///////////////////////////////////////////////////////////////////////////////////////
// ---   Formateo del Evento de Estado del Dispositivo
// ---   * Mirar si hay sitio para generar el nuevo evento
// ---       * Inicializo NumBytes y Puntero al DB de Eventos Generados
// ---       * Calcula el tamaño de bytes que hay en el DB de Eventos Generados
// ---       * Comprobar si hay sitio para un evento más
// ---   *  Formatear el evento de Estado de Inicio de Bucle  INI!
///////////////////////////////////////////////////////////////////////////////////////


///////////////////////////////////////////////////////////////////////////////////////
// --- Mirar si hay sitio para generar un evento más
      L     0;
      T     #NumBytes;  // Inicializo el numero de Bytes
      T     #P_Eventos;  // Inicializo el puntero de Eventos Generados

Inicio_BusquedaFinalEventos_MckeysEnMesa:NOP   0;
      OPN   DB [#DBEventos];  // Calcula el tamaño de bytes que hay en el DB
      L     DBB [#P_Eventos];
      L     0;
      ==I;
      JC    Fin_BusquedaFinalEventos_MckeysEnMesa;  // Buscamos el final del DB = 0

      OPN   DB [#DBEventos];
      L     DBB [#P_Eventos];
      L     ' ';
      ==I;
      JC    Fin_BusquedaFinalEventos_MckeysEnMesa;  // Buscamos el final del DB = ' '

      L     #P_Eventos;  // Incremento de P#1.0
      L     P#1.0;
      +D;
      T     #P_Eventos;

      JU    Inicio_BusquedaFinalEventos_MckeysEnMesa;  // Continuar con el siguiente posicion

Fin_BusquedaFinalEventos_MckeysEnMesa:NOP   0;
      L     #P_Eventos;  // Sacamos el NumBytes Escritos
      SRD   3;
      T     #NumBytes;

      L     #NumBytes;  // Miramos si hay sitio
      L     #MaxBytes;  // Max. que se pueden emitir, parametro
      >I;
      JC    FinalFuncion;  // No se pueden generar más eventos



///////////////////////////////////////////////////////////////////////////////////////
// --- Formatear el evento
      L     #P_Eventos;
      LAR2;  // Puntero al DB de Eventos Generados

      TAR2;  // Mirar si es el primer evento de la lista
      L     0;
      ==I;
      JC    NoEsInicio_ListaDeEventos_MckeysEnMesa;  // Es el primero

      OPN   DB [#DBEventos];
      L     ',';  // Separador entre eventos ','
      T     DBB [AR2, P#0.0];
      +AR2  P#1.0;

NoEsInicio_ListaDeEventos_MckeysEnMesa:NOP   0;

///////////////////////////////////////////////////////////////////////////////
// --- Cuerpo del Evento
      OPN   DB [#DBEventos];  // DB de Eventos Generados (A Emitir)
      L     '{';  // Inicio de Evento '{'
      T     DBB [AR2, P#0.0];
      +AR2  P#1.0;

      L     'CHE!';  // Evento - CHE!
      T     DBD [AR2, P#0.0];
      +AR2  P#4.0;


///////////////////////////////////////////////////////////////////////////////
      L     '[';
      T     DBB [AR2, P#0.0];
      L     'TIPO';
      T     DBD [AR2, P#1.0];
      L     ']';  // Evento - Atributo Mckey '[TIPO]'
      T     DBB [AR2, P#5.0];
      +AR2  P#6.0;

      L     'MESA';
      T     DBD [AR2, P#0.0];
      +AR2  P#4.0;


///////////////////////////////////////////////////////////////////////////////
      OPN   DB [#DBEventos];
      L     '[';  // Evento - Atributo Mesa  '[NUME]'
      T     DBB [AR2, P#0.0];
      L     'NUME';
      T     DBD [AR2, P#1.0];
      L     ']';
      T     DBB [AR2, P#5.0];
      +AR2  P#6.0;

      L     #NumMesa;
      L     "CTE_OffsetMesa";
      +I;
      T     #Valor;

// --- Convertir Valor a ASCII -  Mesa Actual
      TAR2;
      SRD   3;
      T     #NumBytes;  // Miro que offset tiene la String

      CALL  "FC893_Obtener_StringDelAtributo"
      ( DB_String := #NumDBEventos,
        OffsetIni := #NumBytes,
        Valor     := #Valor,
        OffsetFin := #Offset
      );  // Llamo a ObtenerStrinAtributo

      L     #Offset;
      SLD   3;
      LAR2;  // Recupero que offset tiene la String
// --- Ya esta convertido el Valor a ASCI - Fin Mesa Actual



///////////////////////////////////////////////////////////////////////////////
      L     '[';
      T     DBB [AR2, P#0.0];
      L     'OPER';
      T     DBD [AR2, P#1.0];
      L     ']';  // Evento - Atributo Mckey '[TIPO]'
      T     DBB [AR2, P#5.0];
      +AR2  P#6.0;

      L     'MCKY';
      T     DBD [AR2, P#0.0];
      +AR2  P#4.0;


///////////////////////////////////////////////////////////////////////////////
      OPN   DB [#DBEventos];
      L     '[';  // Evento - Atributo Mckeys '[MCKY]'
      T     DBB [AR2, P#0.0];
      L     'MCKY';
      T     DBD [AR2, P#1.0];
      L     ']';
      T     DBB [AR2, P#5.0];
      +AR2  P#6.0;

// ---- Inicio de Mckeys
      OPN   DB [#DBEventos];
      L     '(';
      T     DBB [AR2, P#0.0];
      +AR2  P#1.0;

// --- Bucle de Mckeys >>> Hay Una UT
      L     "DB810_ColasMesas".Colas[#NumMesa].UT_PrimeraMesa;
      T     #NumeroUT;

      SET;  // Hay UT ?
      L     #NumeroUT;
      L     0;
      ==I;
      JC    FinalBucleUTs_MckeysEnMesa;

      L     "DB812_UTs_Control".UT[#NumeroUT].Mckey;
      T     #Valor;

// --- Convertir Valor a ASCII -  Mesa Actual
      TAR2;
      SRD   3;
      T     #NumBytes;  // Miro que offset tiene la String

      CALL  "FC893_Obtener_StringDelAtributo"
      ( DB_String := #NumDBEventos,
        OffsetIni := #NumBytes,
        Valor     := #Valor,
        OffsetFin := #Offset
      );  // Llamo a ObtenerStrinAtributo

      L     #Offset;
      SLD   3;
      LAR2;  // Recupero que offset tiene la String
// --- Ya esta convertido el Valor a ASCI - Fin Mesa Actual

      L     "DB812_UTs_Control".UT[#NumeroUT].UT_SiguienteMesa;
      T     #NumeroUT;

// --- Bucle de Mckeys >>> Hay Mas UTs
IncioBucleUTs_MckeysEnMesa:NOP   0;
      SET;  // Hay UT ?
      L     #NumeroUT;
      L     0;
      ==I;
      JC    FinalBucleUTs_MckeysEnMesa;

      OPN   DB [#DBEventos];
      L     ',';  // Separador de Mckeys
      T     DBB [AR2, P#0.0];
      +AR2  P#1.0;

      L     "DB812_UTs_Control".UT[#NumeroUT].Mckey;
      T     #Valor;

// --- Convertir Valor a ASCII -  Mesa Actual
      TAR2;
      SRD   3;
      T     #NumBytes;  // Miro que offset tiene la String

      CALL  "FC893_Obtener_StringDelAtributo"
      ( DB_String := #NumDBEventos,
        OffsetIni := #NumBytes,
        Valor     := #Valor,
        OffsetFin := #Offset
      );  // Llamo a ObtenerStrinAtributo

      L     #Offset;
      SLD   3;
      LAR2;  // Recupero que offset tiene la String
// --- Ya esta convertido el Valor a ASCI - Fin Mesa Actual


      L     "DB812_UTs_Control".UT[#NumeroUT].UT_SiguienteMesa;
      T     #NumeroUT;
      JU    IncioBucleUTs_MckeysEnMesa;

FinalBucleUTs_MckeysEnMesa:NOP   0;

// --- Final de Mckeys
      OPN   DB [#DBEventos];
      L     ')';
      T     DBB [AR2, P#0.0];
      +AR2  P#1.0;


///////////////////////////////////////////////////////////////////////////////
      OPN   DB [#DBEventos];
      L     '[';  // Evento - Atributo Resultado'[RESU]'
      T     DBB [AR2, P#0.0];
      L     'RESU';
      T     DBD [AR2, P#1.0];
      L     ']';
      T     DBB [AR2, P#5.0];
      +AR2  P#6.0;

      L     'OK';
      T     DBW [AR2, P#0.0];
      +AR2  P#2.0;


///////////////////////////////////////////////////////////////////////////////
// --- Final del Evento

      OPN   DB [#DBEventos];  // DB de Eventos Generados (A Emitir)
      L     '}';  // --- Fin de Evento '}'
      T     DBB [AR2, P#0.0];
      +AR2  P#1.0;


///////////////////////////////////////////////////////////////////////////////
/// -- Dar  por enviado el evento

      SET;
      R     "DB831_Mesas".Mesas[#NumMesa].EventosInformarJdT.MckeysEnMesa;

      JU    Siguiente_BucleDeMesas;



NETWORK
TITLE = Evento de Evento de Todo De Mesa >>> Ocupacion, Mckeys
EnviarEvento_TodoDeMesa:NOP   0;

///////////////////////////////////////////////////////////////////////////////////////
// ---   Formateo del Evento de Estado del Dispositivo
// ---   * Mirar si hay sitio para generar el nuevo evento
// ---       * Inicializo NumBytes y Puntero al DB de Eventos Generados
// ---       * Calcula el tamaño de bytes que hay en el DB de Eventos Generados
// ---       * Comprobar si hay sitio para un evento más
// ---   *  Formatear el evento de Estado de Inicio de Bucle  INI!
///////////////////////////////////////////////////////////////////////////////////////


///////////////////////////////////////////////////////////////////////////////////////
// --- Mirar si hay sitio para generar un evento más
      L     0;
      T     #NumBytes;  // Inicializo el numero de Bytes
      T     #P_Eventos;  // Inicializo el puntero de Eventos Generados

Inicio_BusquedaFinalEventos_TodoDeMesa:NOP   0;
      OPN   DB [#DBEventos];  // Calcula el tamaño de bytes que hay en el DB
      L     DBB [#P_Eventos];
      L     0;
      ==I;
      JC    Fin_BusquedaFinalEventos_TodoDeMesa;  // Buscamos el final del DB = 0

      OPN   DB [#DBEventos];
      L     DBB [#P_Eventos];
      L     ' ';
      ==I;
      JC    Fin_BusquedaFinalEventos_TodoDeMesa;  // Buscamos el final del DB = ' '

      L     #P_Eventos;  // Incremento de P#1.0
      L     P#1.0;
      +D;
      T     #P_Eventos;

      JU    Inicio_BusquedaFinalEventos_TodoDeMesa;  // Continuar con el siguiente posicion

Fin_BusquedaFinalEventos_TodoDeMesa:NOP   0;
      L     #P_Eventos;  // Sacamos el NumBytes Escritos
      SRD   3;
      T     #NumBytes;

      L     #NumBytes;  // Miramos si hay sitio
      L     #MaxBytes;  // Max. que se pueden emitir, parametro
      >I;
      JC    FinalFuncion;  // No se pueden generar más eventos



///////////////////////////////////////////////////////////////////////////////////////
// --- Formatear el evento
      L     #P_Eventos;
      LAR2;  // Puntero al DB de Eventos Generados

      TAR2;  // Mirar si es el primer evento de la lista
      L     0;
      ==I;
      JC    NoEsInicio_ListaDeEventos_TodoDeMesa;  // Es el primero

      OPN   DB [#DBEventos];
      L     ',';  // Separador entre eventos ','
      T     DBB [AR2, P#0.0];
      +AR2  P#1.0;

NoEsInicio_ListaDeEventos_TodoDeMesa:NOP   0;

///////////////////////////////////////////////////////////////////////////////
// --- Cuerpo del Evento
      OPN   DB [#DBEventos];  // DB de Eventos Generados (A Emitir)
      L     '{';  // Inicio de Evento '{'
      T     DBB [AR2, P#0.0];
      +AR2  P#1.0;

      L     'CHE!';  // Evento - CHE!
      T     DBD [AR2, P#0.0];
      +AR2  P#4.0;


///////////////////////////////////////////////////////////////////////////////
      L     '[';
      T     DBB [AR2, P#0.0];
      L     'TIPO';
      T     DBD [AR2, P#1.0];
      L     ']';  // Evento - Atributo Mckey '[TIPO]'
      T     DBB [AR2, P#5.0];
      +AR2  P#6.0;

      L     'MESA';
      T     DBD [AR2, P#0.0];
      +AR2  P#4.0;


///////////////////////////////////////////////////////////////////////////////
      OPN   DB [#DBEventos];
      L     '[';  // Evento - Atributo Mesa  '[NUME]'
      T     DBB [AR2, P#0.0];
      L     'NUME';
      T     DBD [AR2, P#1.0];
      L     ']';
      T     DBB [AR2, P#5.0];
      +AR2  P#6.0;

      L     #NumMesa;
      L     "CTE_OffsetMesa";
      +I;
      T     #Valor;

// --- Convertir Valor a ASCII -  Mesa Actual
      TAR2;
      SRD   3;
      T     #NumBytes;  // Miro que offset tiene la String

      CALL  "FC893_Obtener_StringDelAtributo"
      ( DB_String := #NumDBEventos,
        OffsetIni := #NumBytes,
        Valor     := #Valor,
        OffsetFin := #Offset
      );  // Llamo a ObtenerStrinAtributo

      L     #Offset;
      SLD   3;
      LAR2;  // Recupero que offset tiene la String
// --- Ya esta convertido el Valor a ASCI - Fin Mesa Actual



///////////////////////////////////////////////////////////////////////////////
      L     '[';
      T     DBB [AR2, P#0.0];
      L     'OPER';
      T     DBD [AR2, P#1.0];
      L     ']';  // Evento - Atributo Mckey '[TIPO]'
      T     DBB [AR2, P#5.0];
      +AR2  P#6.0;

      L     'TODO';
      T     DBD [AR2, P#0.0];
      +AR2  P#4.0;


///////////////////////////////////////////////////////////////////////////////
      OPN   DB [#DBEventos];
      L     '[';  // Evento - Atributo Mckeys '[MCKY]'
      T     DBB [AR2, P#0.0];
      L     'MCKY';
      T     DBD [AR2, P#1.0];
      L     ']';
      T     DBB [AR2, P#5.0];
      +AR2  P#6.0;

// ---- Inicio de Mckeys
      OPN   DB [#DBEventos];
      L     '(';
      T     DBB [AR2, P#0.0];
      +AR2  P#1.0;

// --- Bucle de Mckeys >>> Hay Una UT
      L     "DB810_ColasMesas".Colas[#NumMesa].UT_PrimeraMesa;
      T     #NumeroUT;

      SET;  // Hay UT ?
      L     #NumeroUT;
      L     0;
      ==I;
      JC    FinalBucleUTs_TodoDeMesa;

      L     "DB812_UTs_Control".UT[#NumeroUT].Mckey;
      T     #Valor;

// --- Convertir Valor a ASCII -  Mesa Actual
      TAR2;
      SRD   3;
      T     #NumBytes;  // Miro que offset tiene la String

      CALL  "FC893_Obtener_StringDelAtributo"
      ( DB_String := #NumDBEventos,
        OffsetIni := #NumBytes,
        Valor     := #Valor,
        OffsetFin := #Offset
      );  // Llamo a ObtenerStrinAtributo

      L     #Offset;
      SLD   3;
      LAR2;  // Recupero que offset tiene la String
// --- Ya esta convertido el Valor a ASCI - Fin Mesa Actual

      L     "DB812_UTs_Control".UT[#NumeroUT].UT_SiguienteMesa;
      T     #NumeroUT;

// --- Bucle de Mckeys >>> Hay Mas UTs
IncioBucleUTs_TodoDeMesa:NOP   0;
      SET;  // Hay UT ?
      L     #NumeroUT;
      L     0;
      ==I;
      JC    FinalBucleUTs_TodoDeMesa;

      OPN   DB [#DBEventos];
      L     ',';  // Separador de Mckeys
      T     DBB [AR2, P#0.0];
      +AR2  P#1.0;

      L     "DB812_UTs_Control".UT[#NumeroUT].Mckey;
      T     #Valor;

// --- Convertir Valor a ASCII -  Mesa Actual
      TAR2;
      SRD   3;
      T     #NumBytes;  // Miro que offset tiene la String

      CALL  "FC893_Obtener_StringDelAtributo"
      ( DB_String := #NumDBEventos,
        OffsetIni := #NumBytes,
        Valor     := #Valor,
        OffsetFin := #Offset
      );  // Llamo a ObtenerStrinAtributo

      L     #Offset;
      SLD   3;
      LAR2;  // Recupero que offset tiene la String
// --- Ya esta convertido el Valor a ASCI - Fin Mesa Actual


      L     "DB812_UTs_Control".UT[#NumeroUT].UT_SiguienteMesa;
      T     #NumeroUT;
      JU    IncioBucleUTs_TodoDeMesa;

FinalBucleUTs_TodoDeMesa:NOP   0;





// --- Final de Mckeys
      OPN   DB [#DBEventos];
      L     ')';
      T     DBB [AR2, P#0.0];
      +AR2  P#1.0;


///////////////////////////////////////////////////////////////////////////////
      OPN   DB [#DBEventos];
      L     '[';  // Evento - Atributo Ocupacion '[OCUP]'
      T     DBB [AR2, P#0.0];
      L     'OCUP';
      T     DBD [AR2, P#1.0];
      L     ']';
      T     DBB [AR2, P#5.0];
      +AR2  P#6.0;

      L     'NO';  // No Ocupado

      SET;
      AN    "DB900_Estado_Mesas".EstadoVI[#NumMesa].En_PHS_1;
      AN    "DB900_Estado_Mesas".EstadoVI[#NumMesa].En_PHS_2;
      JC    NoOcupado_TodoDeMesa;

      L     'SI';  // Esta Ocupado

NoOcupado_TodoDeMesa:NOP   0;
      OPN   DB [#DBEventos];
      T     DBW [AR2, P#0.0];
      +AR2  P#2.0;


///////////////////////////////////////////////////////////////////////////////
      OPN   DB [#DBEventos];
      L     '[';  // Evento - Atributo Resultado'[RESU]'
      T     DBB [AR2, P#0.0];
      L     'RESU';
      T     DBD [AR2, P#1.0];
      L     ']';
      T     DBB [AR2, P#5.0];
      +AR2  P#6.0;

      L     'OK';
      T     DBW [AR2, P#0.0];
      +AR2  P#2.0;


///////////////////////////////////////////////////////////////////////////////
// --- Final del Evento

      OPN   DB [#DBEventos];  // DB de Eventos Generados (A Emitir)
      L     '}';  // --- Fin de Evento '}'
      T     DBB [AR2, P#0.0];
      +AR2  P#1.0;


///////////////////////////////////////////////////////////////////////////////
/// -- Dar  por enviado el evento

      SET;
      R     "DB831_Mesas".Mesas[#NumMesa].EventosInformarJdT.TodoDeMesa;

      JU    Siguiente_BucleDeMesas;



NETWORK
TITLE = Emision de Evento Rearme
EnviarEvento_rearme:NOP   0;

///////////////////////////////////////////////////////////////////////////////////////
// ---   Formateo del Evento de Estado del Dispositivo
// ---   * Mirar si hay sitio para generar el nuevo evento
// ---       * Inicializo NumBytes y Puntero al DB de Eventos Generados
// ---       * Calcula el tamaño de bytes que hay en el DB de Eventos Generados
// ---       * Comprobar si hay sitio para un evento más
// ---   *  Formatear el evento de Estado de Inicio de Bucle
///////////////////////////////////////////////////////////////////////////////////////

// --- Primero miramos si tenemos configurado emitir el evento o no
      SET;
      A     "DB831_Mesas".Mesas[#NumMesa].EventosInformarJdT.Evento_Rearme;
      JC    emite_evento_rearme;

      SET;
      R     "DB831_Mesas".Mesas[#NumMesa].Memorias.Evento_rearme;
      JC    Siguiente_BucleDeMesas;

///////////////////////////////////////////////////////////////////////////////////////
// --- Mirar si hay sitio para generar un evento más
emite_evento_rearme:NOP   0;
      L     0;
      T     #NumBytes;  // Inicializo el numero de Bytes
      T     #P_Eventos;  // Inicializo el puntero de Eventos Generados

Inicio_BusquedaFinalEventos_rearme:NOP   0;
      OPN   DB [#DBEventos];  // Calcula el tamaño de bytes que hay en el DB
      L     DBB [#P_Eventos];
      L     0;
      ==I;
      JC    Fin_BusquedaFinalEventos_rearme;  // Buscamos el final del DB = 0

      OPN   DB [#DBEventos];
      L     DBB [#P_Eventos];
      L     ' ';
      ==I;
      JC    Fin_BusquedaFinalEventos_rearme;  // Buscamos el final del DB = ' '

      L     #P_Eventos;  // Incremento de P#1.0
      L     P#1.0;
      +D;
      T     #P_Eventos;

      JU    Inicio_BusquedaFinalEventos_rearme;  //Continuar con el siguiente posicion

Fin_BusquedaFinalEventos_rearme:NOP   0;
      L     #P_Eventos;  // Sacamos el NumBytes Escritos
      SRD   3;
      T     #NumBytes;

      L     #NumBytes;  // Miramos si hay sitio
      L     #MaxBytes;  // Max. que se pueden emitir, parametro
      >I;
      JC    FinalFuncion;  // No se pueden generar más eventos



///////////////////////////////////////////////////////////////////////////////////////
// --- Formatear el evento
      L     #P_Eventos;
      LAR2;  // Puntero al DB de Eventos Generados

      TAR2;  // Mirar si es el primer evento de la lista
      L     0;
      ==I;
      JC    NoEsInicio_ListaDeEventos_rearme;  // Es el primero

      OPN   DB [#DBEventos];
      L     ',';  // Separador entre eventos ','
      T     DBB [AR2, P#0.0];
      +AR2  P#1.0;

NoEsInicio_ListaDeEventos_rearme:NOP   0;

///////////////////////////////////////////////////////////////////////////////
// --- Cuerpo del Evento
      OPN   DB [#DBEventos];  // DB de Eventos Generados (A Emitir)
      L     '{';  // Inicio de Evento '{'
      T     DBB [AR2, P#0.0];
      +AR2  P#1.0;

      L     'EVEN';  // Evento - EVEN
      T     DBD [AR2, P#0.0];
      +AR2  P#4.0;


///////////////////////////////////////////////////////////////////////////////
      L     '[';
      T     DBB [AR2, P#0.0];
      L     'TIPO';
      T     DBD [AR2, P#1.0];
      L     ']';  // Evento - Atributo Mckey '[TIPO]'
      T     DBB [AR2, P#5.0];
      +AR2  P#6.0;

      L     'MESA';
      T     DBD [AR2, P#0.0];
      +AR2  P#4.0;


///////////////////////////////////////////////////////////////////////////////
      OPN   DB [#DBEventos];
      L     '[';  // Evento - Atributo Mesa  '[NUME]'
      T     DBB [AR2, P#0.0];
      L     'NUME';
      T     DBD [AR2, P#1.0];
      L     ']';
      T     DBB [AR2, P#5.0];
      +AR2  P#6.0;

      L     #NumMesa;
      L     "CTE_OffsetMesa";
      +I;
      T     #Valor;

// --- Convertir Valor a ASCII -  Mesa Actual
      TAR2;
      SRD   3;
      T     #NumBytes;  // Miro que offset tiene la String

      CALL  "FC893_Obtener_StringDelAtributo"
      ( DB_String := #NumDBEventos,
        OffsetIni := #NumBytes,
        Valor     := #Valor,
        OffsetFin := #Offset
      );  // Llamo a ObtenerStrinAtributo

      L     #Offset;
      SLD   3;
      LAR2;  // Recupero que offset tiene la String
// --- Ya esta convertido el Valor a ASCI - Fin Mesa Actual



///////////////////////////////////////////////////////////////////////////////
      L     '[';
      T     DBB [AR2, P#0.0];
      L     'OPER';
      T     DBD [AR2, P#1.0];
      L     ']';  // Evento - Atributo Mckey '[TIPO]'
      T     DBB [AR2, P#5.0];
      +AR2  P#6.0;

      L     'REAR';
      T     DBD [AR2, P#0.0];
      +AR2  P#4.0;


///////////////////////////////////////////////////////////////////////////////
// --- Final del Evento

      OPN   DB [#DBEventos];  // DB de Eventos Generados (A Emitir)
      L     '}';  // --- Fin de Evento '}'
      T     DBB [AR2, P#0.0];
      +AR2  P#1.0;


///////////////////////////////////////////////////////////////////////////////
/// -- Dar  por enviado el evento

      SET;
      R     "DB831_Mesas".Mesas[#NumMesa].Memorias.Evento_rearme;

      JU    Siguiente_BucleDeMesas;



NETWORK
TITLE = Final de la Función
/////////////////////////////////////////////////////////////////////////////////////
FinalFuncion:NOP   0;


END_FUNCTION

FUNCTION "FC700_JDT02ControlTracking" : Void   // FC700, LAD
{ S7_Optimized_Access := 'FALSE' }
AUTHOR : TRACKING
NAME : 20141014
VERSION : 4.0
// stored: AutoNumber false, SetENOAutomatically false
BEGIN

NETWORK
TITLE = Previo
// -----------------------------------------------------------------------
// --- Inicialializacion
// --- Borrado de la Base de Datosç

      CALL  "FC701_JDT02ControlCOM";  // Control del Puerto
      CALL  "FC706_JDT02Borrado";



NETWORK
TITLE = Control del Sistema
// ---------------------------------------------------------------------
// --- Control de Recepcion de Eventos

      CALL  "FC702_JDT02RecJdTMensaje";
      CALL  "FC704_JDT02AnalisisRecibidos";
      CALL  "FC810_EventosRecibidos"
      ( NumJDT := 2
      );


// ---------------------------------------------------------------------
// --- Control de EmisionEventos de Eventos

      CALL  "FC811_EventosGenerados"
      ( NumJdT := 2
      );
      CALL  "FC705_JDT02AnalisisEnviados";
      CALL  "FC703_JDT02EmiJdTMensaje";


// ---------------------------------------------------------------------
// --- Control de EmisionEventos de Router
//     *  Proceso Inicialización bucle
//     *  Eventos de la Pantalla (Movimientos)
//     *  Eventos de Reset V2.0   >>> 2023 01 05

//      CALL  "FC816_EventosEnv_Router"
//         NumJDT :=2

// NIEVES 10/04/25
      CALL  "FC717_Emision_Routing"
      ( NumJDT := 2
      );


      CALL  "FC815_EventosEnv_Control"
      ( NumJDT := 2
      );
      CALL  "FC817_EventosEnv_Reset"
      ( NumJDT := 2
      );


Fin:  NOP   0;


END_FUNCTION

FUNCTION "FC701_JDT02ControlCOM" : Void   // FC701, LAD
TITLE = "ControlCOM" - Control de Comunicaciones
{ S7_Optimized_Access := 'FALSE' }
AUTHOR : TRACKING
NAME : 20150129
VERSION : 3.1
// - Contorol y valida el Enlace entre el PLC y el PC
// - Varible: EnlaceCP_OK
// stored: AutoNumber false, SetENOAutomatically false
   VAR_TEMP
      Temporal : Struct   // Temporal para el tratamiento de Result 01
         "0.0" : Bool;
         "0.1" : Bool;
         "0.2" : Bool;
         "0.3" : Bool;
         "0.4" : Bool;
         "0.5" : Bool;
         "0.6" : Bool;
         "0.7" : Bool;
         "1.0" : Bool;
         "1.1" : Bool;
         "1.2" : Bool;
         "1.3" : Bool;
         "1.4" : Bool;
         "1.5" : Bool;
         "1.6" : Bool;
         "1.7" : Bool;
         "2.0" : Bool;
         "2.1" : Bool;
         "2.2" : Bool;
         "2.3" : Bool;
         "2.4" : Bool;
         "2.5" : Bool;
         "2.6" : Bool;
         "2.7" : Bool;
         "3.0" : Bool;
         "3.1" : Bool;
         "3.2" : Bool;
         "3.4" : Bool;
         "3.5" : Bool;
         "3.6" : Bool;
         "3.7" : Bool;
      END_STRUCT;
      P_Temporal : DWord;
      TMPEnlace_OK : Bool;
   END_VAR
BEGIN

NETWORK
TITLE = Control del Enlace - Puerto 2001
// - Distribución  - Conexion  - Desconesion  - Final    ------------------------------------------------------------------------------------------------------   Control del Enlace - Distribución   --- Si hay que desconetar   --- Si esta conectado
      A     "DB701_JDT02StatusCOM".CNTRL_Reset;  // Si hay que desconectar
      O     "DB701_JDT02StatusCOM".RecJdT_Reset;
      O     "DB701_JDT02StatusCOM".EmiJdT_Reset;
      JC    DesConectar;

      A     "DB701_JDT02StatusCOM".EnlaceCP_OK;  // Si está conectado
      JC    Final;

      JU    Conectar;  // Hay que conectar

// ------------------------------------------------------------------------------------------------------
// Control del Enlace - Conexion
// --- Mirar si hay que activar Flanco
// --- Mirar si hay petición de conexion activa
// --- Llamada de Conexion
// --- Comprobación de la Conexion

Conectar:NOP   0;
      AN    "DB891_VariablesTCP".TCON_JdT_PLC_Busy_JDT02;
      AN    "DB891_VariablesTCP".TCON_JdT_PLC_Req_JDT02;
      AN    "DB891_VariablesTCP".TCON_JdT_PLC_Flanco_JDT02;
      =     "DB891_VariablesTCP".TCON_JdT_PLC_Flanco_JDT02;  // -- Activar flanco

      A     "DB891_VariablesTCP".TCON_JdT_PLC_Flanco_JDT02;
      AN    "DB891_VariablesTCP".TCON_JdT_PLC_Req_JDT02;
      S     "DB891_VariablesTCP".TCON_JdT_PLC_Req_JDT02;
      R     "DB891_VariablesTCP".TDISCON_JdT_PLC_Req_JDT02;  // -- Petición de Conexion Activa

      CALL  TCON, "DB896_TCON_JdT_PLC_JDT02"
      ( REQ     := "DB891_VariablesTCP".TCON_JdT_PLC_Flanco_JDT02,
        ID      := W#16#3,
        DONE    := "DB891_VariablesTCP".TCON_JdT_PLC_Done_JDT02,
        BUSY    := "DB891_VariablesTCP".TCON_JdT_PLC_Busy_JDT02,
        ERROR   := "DB891_VariablesTCP".TCON_JdT_PLC_Error_JDT02,
        STATUS  := "DB891_VariablesTCP".TCON_JdT_PLC_Status_JDT02,
        CONNECT := "DB700_JDTD02ConfigEnlace"
      );


      A     "DB891_VariablesTCP".TCON_JdT_PLC_Done_JDT02;  // -- Comprobacion de la Conexion
      R     "DB891_VariablesTCP".TCON_JdT_PLC_Req_JDT02;
      S     "DB701_JDT02StatusCOM".EnlaceCP_OK;

      A     "DB891_VariablesTCP".TCON_JdT_PLC_Error_JDT02;  // -- Error en conexion
      R     "DB891_VariablesTCP".TCON_JdT_PLC_Req_JDT02;

      A     "DB891_VariablesTCP".TCON_JdT_PLC_Req_JDT02;  // --- Control de Bloqueo
      AN    "DB891_VariablesTCP".TCON_JdT_PLC_Busy_JDT02;
      R     "DB891_VariablesTCP".TCON_JdT_PLC_Req_JDT02;

      JU    Final;  // Fin de la Conexión

// ------------------------------------------------------------------------------------------------------
// Control del Enlace - Desconexion
// --- Mirar si hay que activar Flanco
// --- Mirar si hay petición de desconexion activa
// --- Llamada de DesConexion
// --- Comprobación de la DesConexion

DesConectar:SET;
      R     "DB701_JDT02StatusCOM".EnlaceCP_OK;

      AN    "DB891_VariablesTCP".TDISCON_JdT_PLC_Busy_JDT02;
      AN    "DB891_VariablesTCP".TDISCON_JdT_PLC_Req_JDT02;
      AN    "DB891_VariablesTCP".TDISCON_JdT_PLC_Flanco_JDT02;
      =     "DB891_VariablesTCP".TDISCON_JdT_PLC_Flanco_JDT02;  // -- Activar Flanco


      A     "DB891_VariablesTCP".TDISCON_JdT_PLC_Flanco_JDT02;
      AN    "DB891_VariablesTCP".TDISCON_JdT_PLC_Req_JDT02;
      S     "DB891_VariablesTCP".TDISCON_JdT_PLC_Req_JDT02;
      R     "DB891_VariablesTCP".TCON_JdT_PLC_Req_JDT02;  // -- Petición de DesConexion Activa

      CALL  TDISCON, "DB897_TDISCON_JdT_PLC_JDT02"
      ( REQ    := "DB891_VariablesTCP".TDISCON_JdT_PLC_Flanco_JDT02,
        ID     := W#16#3,
        DONE   := "DB891_VariablesTCP".TDISCON_JdT_PLC_Done_JDT02,
        BUSY   := "DB891_VariablesTCP".TDISCON_JdT_PLC_Busy_JDT02,
        ERROR  := "DB891_VariablesTCP".TDISCON_JdT_PLC_Error_JDT02,
        STATUS := "DB891_VariablesTCP".TDISCON_JdT_PLC_Status_JDT02
      );



      A     "DB891_VariablesTCP".TDISCON_JdT_PLC_Done_JDT02;  // -- Comprobacion de la DesConexión
      R     "DB891_VariablesTCP".TDISCON_JdT_PLC_Req_JDT02;


      R     "DB701_JDT02StatusCOM".CNTRL_Reset;
      R     "DB701_JDT02StatusCOM".RecJdT_Reset;
      R     "DB701_JDT02StatusCOM".EmiJdT_Reset;

      A     "DB891_VariablesTCP".TDISCON_JdT_PLC_Error_JDT02;  // -- Error en la DesConexion
      R     "DB891_VariablesTCP".TDISCON_JdT_PLC_Req_JDT02;

      O(;
      L     "DB891_VariablesTCP".TDISCON_JdT_PLC_Status_JDT02;
      L     W#16#80A3;  //Se está intentando deshacer una conexión no existente
      ==I;
      );
      O(;
      L     "DB891_VariablesTCP".TDISCON_JdT_PLC_Status_JDT02;
      L     W#16#8086;  //El parámetro ID se encuentra en un rango no permitido
      ==I;
      );
      R     "DB891_VariablesTCP".TDISCON_JdT_PLC_Busy_JDT02;
      R     "DB891_VariablesTCP".TDISCON_JdT_PLC_Req_JDT02;
      R     "DB891_VariablesTCP".TDISCON_JdT_PLC_Flanco_JDT02;

      A     "DB891_VariablesTCP".TDISCON_JdT_PLC_Req_JDT02;  // --- Control de Bloqueo
      AN    "DB891_VariablesTCP".TDISCON_JdT_PLC_Busy_JDT02;
      R     "DB891_VariablesTCP".TDISCON_JdT_PLC_Req_JDT02;

      R     "DB701_JDT02StatusCOM".CNTRL_Reset;
      R     "DB701_JDT02StatusCOM".RecJdT_Reset;
      R     "DB701_JDT02StatusCOM".EmiJdT_Reset;

      JU    Final;  // Fin de la DesConexión

// ------------------------------------------------------------------------------------------------------
// Control del Enlace - Final

Final:NOP   0;


END_FUNCTION

FUNCTION "FC706_JDT02Borrado" : Void   // FC706, LAD
TITLE = "BorrodoTracking" - Borrado de toda la Base de Datos
{ S7_Optimized_Access := 'FALSE' }
AUTHOR : TRACKING
NAME : 20130301
VERSION : 3.0
// - Borrado de todos los DB's
// - Inicializadcion del DB de DatosUT
// stored: AutoNumber false, SetENOAutomatically false
   VAR_TEMP
      NumeroUT : Int;
      NumDB : Word;
      UTVacia : Int;
   END_VAR
BEGIN

NETWORK
TITLE = Borrado de todos los DB's de Comunicacion
// -------------------------------------------------------------------------------
// --- Mirar si hay que resetear
      AN    "DB701_JDT02StatusCOM".ResetBD;
      JC    NoResetear;

// -------------------------------------------------------------------------------
// Borrado de los DB de Recepcion de Eventos

      CALL  "FC898_BorrarMensaje"
      ( DB_A_RESET := "DB702_JDT02RecepMensaje"
      );
      CALL  "FC898_BorrarMensaje"
      ( DB_A_RESET := "DB704_JDT02UltimoRecibido"
      );
      CALL  "FC898_BorrarMensaje"
      ( DB_A_RESET := "DB708_JDT02EventosRecibidos"
      );

// -------------------------------------------------------------------------------
// Borrado de los DB de Emision de Eventos

      CALL  "FC898_BorrarMensaje"
      ( DB_A_RESET := "DB703_JDT02EmisionMensaje"
      );
      CALL  "FC898_BorrarMensaje"
      ( DB_A_RESET := "DB705_JDT02UltimoEnviado"
      );
      CALL  "FC898_BorrarMensaje"
      ( DB_A_RESET := "DB706_JDT02EmisionAK"
      );
      CALL  "FC898_BorrarMensaje"
      ( DB_A_RESET := "DB707_JDT02EventosGenerados"
      );

// -------------------------------------------------------------------------------
// Borrado de los DB de la BD de Mesas
// El DB de CrucesMesas no se borra, esto es fijo para cada instalación

      CALL  "FC898_BorrarMensaje"
      ( DB_A_RESET := "DB810_ColasMesas"
      );
      CALL  "FC898_BorrarMensaje"
      ( DB_A_RESET := "DB811_ColasMckeys"
      );

      CALL  "FC898_BorrarMensaje"
      ( DB_A_RESET := "DB812_UTs_Control"
      );
      CALL  "FC898_BorrarMensaje"
      ( DB_A_RESET := "DB813_UTs_Ruta"
      );

      CALL  "FC898_BorrarMensaje"
      ( DB_A_RESET := "DB814_UTs_Etiqueta"
      );
      CALL  "FC898_BorrarMensaje"
      ( DB_A_RESET := "DB815_UTs_Datos"
      );
      CALL  "FC898_BorrarMensaje"
      ( DB_A_RESET := "DB816_UTs_TextoPantalla"
      );
      CALL  "FC898_BorrarMensaje"
      ( DB_A_RESET := "DB820_UTs_DatosQUBIQA"
      );
      CALL  "FC898_BorrarMensaje"
      ( DB_A_RESET := "DB821_UTs_DatosIKPAL"
      );


// -------------------------------------------------------------------------------
// Borrado de los DB de la BD de Dispositivos

      CALL  "FC898_BorrarMensaje"
      ( DB_A_RESET := "DB830_Dispositivos"
      );
      CALL  "FC898_BorrarMensaje"
      ( DB_A_RESET := "DB831_Mesas"
      );
      CALL  "FC898_BorrarMensaje"
      ( DB_A_RESET := "DB832_Maquinas"
      );


// -------------------------------------------------------------------------------
// Borrado de los DB Emision y Recepcion con la instalación

      CALL  "FC898_BorrarMensaje"
      ( DB_A_RESET := "DB840_Emision"
      );
      CALL  "FC898_BorrarMensaje"
      ( DB_A_RESET := "DB841_Recepcion"
      );
      CALL  "FC898_BorrarMensaje"
      ( DB_A_RESET := "DB843_RecepcionPantalla"
      );

      SET;
      R     "DB701_JDT02StatusCOM".ResetBD;

      JU    FinFuncion;  // El siguiente segmento no se realiza


NETWORK
TITLE = ----
// Se acabo la inicializacion
NoResetear:NOP   0;
      L     0;
      LAR1;

// -------------------------------------------------------------------------------
// Borrado de los DB de Recepcion de Eventos, si es necesario

      OPN   "DB702_JDT02RecepMensaje";
      L     DBB [AR1, P#0.0];
      L     ' ';
      <>I;
      JC    S_31;
      CALL  "FC898_BorrarMensaje"
      ( DB_A_RESET := "DB702_JDT02RecepMensaje"
      );

S_31: OPN   "DB704_JDT02UltimoRecibido";
      L     DBB [AR1, P#0.0];
      L     ' ';
      <>I;
      JC    S_32;
      CALL  "FC898_BorrarMensaje"
      ( DB_A_RESET := "DB704_JDT02UltimoRecibido"
      );

S_32: OPN   "DB708_JDT02EventosRecibidos";
      L     DBB [AR1, P#0.0];

      L     ' ';
      <>I;
      JC    S_33;
      CALL  "FC898_BorrarMensaje"
      ( DB_A_RESET := "DB708_JDT02EventosRecibidos"
      );

// -------------------------------------------------------------------------------
// Borrado de los DB de Emision de Eventos, si es necesario

S_33: OPN   "DB703_JDT02EmisionMensaje";
      L     DBB [AR1, P#0.0];
      L     ' ';
      <>I;
      JC    S_34;
      CALL  "FC898_BorrarMensaje"
      ( DB_A_RESET := "DB703_JDT02EmisionMensaje"
      );

S_34: OPN   "DB705_JDT02UltimoEnviado";
      L     DBB [AR1, P#0.0];
      L     ' ';
      <>I;
      JC    S_35;
      CALL  "FC898_BorrarMensaje"
      ( DB_A_RESET := "DB705_JDT02UltimoEnviado"
      );

S_35: OPN   "DB706_JDT02EmisionAK";
      L     DBB [AR1, P#0.0];
      L     ' ';
      <>I;
      JC    S_36;
      CALL  "FC898_BorrarMensaje"
      ( DB_A_RESET := "DB706_JDT02EmisionAK"
      );

S_36: OPN   "DB707_JDT02EventosGenerados";
      L     DBB [AR1, P#0.0];
      L     ' ';
      <>I;
      JC    S_39;
      CALL  "FC898_BorrarMensaje"
      ( DB_A_RESET := "DB707_JDT02EventosGenerados"
      );

S_39: NOP   0;
      JU    FinFuncion;


NETWORK
TITLE = Final de la funcion
FinFuncion:NOP   0;



END_FUNCTION

FUNCTION "FC704_JDT02AnalisisRecibidos" : Void   // FC704, LAD
TITLE = "AnalisisRecibidos" - Analizar los mensajes recibidos por TCP/IP
{ S7_Optimized_Access := 'FALSE' }
AUTHOR : TRACKING
NAME : 20141014
VERSION : 4.0
// - Analizar si el mensaje en si es correcto
// - Distribución
//    - Mensaje ACKN (Validar ID)
//    - Mensaje PING
//    - Resto de mensajes (Validar ID)
// stored: AutoNumber false, SetENOAutomatically false
   VAR_TEMP
      Longitud : UDInt;   // Longitud del Mensaje
      IDMensaje : UDInt;   // ID del Mensaje Recibido
      IniListaEventos : DWord;   // Puntero donde empieza la lista de los eventos
      BytesListaEventos : UDInt;   // Numero de bytes que tiene la lista de los eventos
      DBUltimoRec : Word;   // DB del Ultimo Mensaje Recibido
      DBUltimoEmi : Word;   // DB del Ultimo Mensaje Enviado
      DBEventosRec : Word;   // DB de lista de Eventos Recibidos
      DBEmiAK : Word;   // DB de Emision del Evento AK - Confirmacion
      ReturnValor : Int;   // Temporal
      POrigen : Any;   // Puntero ANY del Origen
      PDestino : Any;   // Puntero ANY del Destino
      IdentEmisor : DWord;
      IdentReceptor : DWord;
      TMPEsperaKA : UDInt;
   END_VAR
BEGIN

NETWORK
TITLE = Inicializamos
// - Inicializaciones de las variables de los DB
// - Coger de la configuracion el Identificador del Emisor (12)
// - Coger de la configuracion el Identificador del Receptor (18)
// -------------------------------------------------------------------------------------------
// Si trabaja sin Agencia  2018 01 24
      SET;
      AN    "Activar_JDT02";  // Mirar si se trabaja con agencia
      JC    Final;

// --------------------------------------------------------------------------------------------
// Inicializaciones de las variables de los DB

      L     "JDT2_NDB_UltimoRec";  // Cogemos el DB de UltimoRecibido
      T     #DBUltimoRec;
      L     "JDT2_NDB_EventosRec";  // Cogemos el DB de EventosRecibidos
      T     #DBEventosRec;

      L     "JDT2_NDB_AKEmi";  // Cogemos el DB de EmisionAK
      T     #DBEmiAK;
      L     "JDT2_NDB_UltimoEmi";  // Cogemos el DB de UltimoEnviado
      T     #DBUltimoEmi;


// --------------------------------------------------------------------------------------------
// Coger de la configuracion el Idendificador del emisor

      L     "JDT2_IdentEmisor";
      T     #IdentEmisor;

// --------------------------------------------------------------------------------------------
// Coger de la configuracion el Idendificador del receptor

      L     "JDT2_IdentReceptor";
      T     #IdentReceptor;


NETWORK
TITLE = Comprobación de la consistencia del mensaje
// Mirar si es correcto
// - Si es Inicio del Mensaje
// - Si es Fin del Mensaje
// - Si es Correcto el Destinario del Mensaje
// - Si es Correcto el Origen del Mensaje
// --------------------------------------------------------------------------------------------
// Mirar si hay mensaje

      L     0;  // Preparar el puntero al Primer byte
      LAR1;
      OPN   DB [#DBUltimoRec];
      L     DBB [AR1, P#0.0];  // Si hay mensaje a tratar <> 0 el primer byte
      L     0;
      ==I;
      JC    Final;  // No hay mensaje

// --------------------------------------------------------------------------------------------
// 1º Paso - Comprobación de que existe Inicio de Mensaje

      OPN   DB [#DBUltimoRec];
      L     DBB [AR1, P#0.0];  // Inicio de Mensaje debe ser 0x02
      L     2;
      ==I;
      JCN   ErrorDeMensajeRecibido;  // Error de Mensaje, Inicio NOK

// --------------------------------------------------------------------------------------------
// 2º Paso - Comprobación de que existe Final del Mensaje

      CALL  "FC890_EtiqChar_EtiqDInt"
      ( DB_String   := "JDT2_NDB_UltimoRec",  // DB del UltimoRecibido
        Long_String := 5,
        Offset_Ini  := 20,
        Valor       := #Longitud
      );  // Calcular la longitud del mensaje

      L     #Longitud;  // Preparar el puntero
      L     1;
      -D;
      SLD   3;
      LAR1;
      OPN   DB [#DBUltimoRec];  // Fin de Mensaje debe ser 0x03
      L     DBB [AR1, P#0.0];
      L     3;
      ==I;
      JCN   ErrorDeMensajeRecibido;  // Error de Mensaje, Fin NOK

// --------------------------------------------------------------------------------------------
// 3º Paso - Comprobación del Emisor del  Mensaje

      L     0;  // Preparar Puntero
      LAR1;
      OPN   DB [#DBUltimoRec];
      L     DBD [AR1, P#6.0];  // Comprobacion del Emisor
      L     #IdentReceptor;
      <>D;
      JC    ErrorDeMensajeRecibido;  // Error de Mensaje, Emisor NOK

// --------------------------------------------------------------------------------------------
// 4º Paso - Comprobación del Receptor del  Mensaje

      OPN   DB [#DBUltimoRec];
      L     DBD [AR1, P#11.0];  // Comprobación del Receptor
      L     #IdentEmisor;
      <>D;
      JC    ErrorDeMensajeRecibido;  // Error de Mensaje, Receptor NOK


NETWORK
TITLE = Distribucion
// - Mirar si es mensaje ACKN - Confirmacion
// - Mirar si es mensaje PING - Keep Alive
// - Es Mensaje de Evento
// --------------------------------------------------------------------------------------------
// 1º Paso - Mirar si es Mensaje AK

      L     0;  // Preparar puntero
      LAR1;
      OPN   DB [#DBUltimoRec];
      L     DBD [AR1, P#24.0];
      L     'ACKN';
      ==I;
      JC    MensajeRecibido_AcuseDeRecibo;  // Recibido Mensaje ACKN - Confirmacion

// --------------------------------------------------------------------------------------------
// 2º Paso - Mirar si es Mensaje KA

      OPN   DB [#DBUltimoRec];
      L     DBD [AR1, P#24.0];
      L     'PING';
      ==I;
      JC    MensajeRecibido_KeepAlive;  // Recibido Mensaje PING - Keep Alive

// --------------------------------------------------------------------------------------------
// 3º Paso - Es Mensaje Evento

      JU    MensajeRecibido_ListaDeEventos;  // Otro tipo de Evento


NETWORK
TITLE = Recibido Mensaje ACKN - Confirmacion del Mensaje Enviado
// - Mirar si esta esperando el Mensaje ACKN - Confirmacion
// - Comprobacion del ID del Mensaje
// - Si es el mismo Numero Secuencial dar por envioado el Mensaje
// - Resetear la variable del Timer Keep Alive y Borrar Mensaje Tratado
// --------------------------------------------------------------------------------------------
// 1º Paso - Comprobamos si esta esperando el Mensaje
MensajeRecibido_AcuseDeRecibo:NOP   0;

      L     0;
      LAR1;
      OPN   DB [#DBUltimoEmi];
      L     DBB [AR1, P#0.0];
      L     'N';  // Mirar si esta esperando que se reciba el AK
      <>I;
      JC    MensajeRecibido_Inesperado;  // No espara el Mensaje AK

// --------------------------------------------------------------------------------------------
// 2º Paso - Comprobamos ID del mensaje

      CALL  "FC890_EtiqChar_EtiqDInt"
      ( DB_String   := "JDT2_NDB_UltimoRec",  // DB del UltimoRecibido
        Long_String := 4,
        Offset_Ini  := 4,
        Valor       := #IDMensaje
      );  // Calcular  el Numero Secuencial

      L     #IDMensaje;  // Si es el mismo Numero Secuencial
      L     "DB701_JDT02StatusCOM".ID_UltimoEnviado;
      <>I;
      JC    MensajeRecibido_Inesperado;  // No es el mismo Numero Secuencial

// --------------------------------------------------------------------------------------------
// 3º Paso - Si es el mismo Numero Secuencial dar por enviado el Mensaje

      SET;
      R     "DB701_JDT02StatusCOM".EsperandoAK;

// nieves Control  reintentos
      L     0;
      T     "Reintentos_JDT2";


// fin control reintentos


      CALL  "FC898_BorrarMensaje"
      ( DB_A_RESET := "DB705_JDT02UltimoEnviado"  // ¿Hay que borrar asi?
      );  // Damos por acabado el envio del mensaje

// --------------------------------------------------------------------------------------------
// 4º Paso - Resetear variable para el Timer de Keep Alive
//         - Borrar Mensaje tratado
MensajeRecibido_Inesperado:NOP   0;

      SET;
      R     "DB701_JDT02StatusCOM".KeepAlive_Recibido;  // Reseteamos el Timer de KeepAlive

      CALL  "FC898_BorrarMensaje"
      ( DB_A_RESET := "DB704_JDT02UltimoRecibido"  // ¿HAy que borrar asi?
      );  // Damos por acabado el mensaje recibido

      JU    Final;


NETWORK
TITLE = Recibido Mensaje PING - Keep Alive
// - Resetear variable que trata el Timer de Keep Alive
// - Borrar Mensaje Tratado

// --------------------------------------------------------------------------------------------
// 1º Paso - Resetear variable para el Timer de Keep Alive
//         - Borrar Mensaje tratado

MensajeRecibido_KeepAlive:NOP   0;

      SET;
      R     "DB701_JDT02StatusCOM".KeepAlive_Recibido;  // Reseteamos el Timer de KeepAlive

      CALL  "FC898_BorrarMensaje"
      ( DB_A_RESET := "DB704_JDT02UltimoRecibido"  // ¿HAy que borrar asi?
      );  // Damos por acabado el envio del mensaje

      JU    Final;

NETWORK
TITLE = Recibido Mensaje de Lista de Eventos
// - Validar el ID del Mensaje Recibido
// - Miramos si se puede tratar el Mensaje de Eventos
// - Copiar la lista de eventos
// --------------------------------------------------------------------------------------------
// 1º Paso - Validar el ID del Mensaje Recibido

MensajeRecibido_ListaDeEventos:NOP   0;

      CALL  "FC890_EtiqChar_EtiqDInt"
      ( DB_String   := "JDT2_NDB_UltimoRec",  // DB del UltimoRecibido
        Long_String := 4,
        Offset_Ini  := 4,
        Valor       := #IDMensaje
      );  // Calcular  el Numero Secuencial

      L     #IDMensaje;  // Comprobar Si el ID = 0
      L     0;
      ==I;
      JC    EINI;

      L     #IDMensaje;  // Comprobar si es el ID Valido
      L     "DB701_JDT02StatusCOM".ID_UltimoRecibido;
      ==I;
      JC    MensajeRecibido_OK;  // No es valido el Numero Secuencial, Enviar ACKN

// --------------------------------------------------------------------------------------------
// 2º Paso - Miramos si se puede tratar el Mensaje de Eventos

EINI: L     0;
      LAR1;
      OPN   DB [#DBEventosRec];
      L     DBB [AR1, P#0.0];  // Vacio - Primer Byte a 0
      L     0;
      <>I;
      JC    Final;  // No puede ser tratado todabia

// --------------------------------------------------------------------------------------------
// 3º Paso - Copiar la lista de eventos

      L     0;  // Preparo el Inicio de la Lista Eventos a Copiar
      LAR1;
      +AR1  P#22.0;
      TAR1;
      T     #IniListaEventos;

      L     #Longitud;  // Numero de Bytes de la Lista de Eventos a Copiar
      L     22;
      -D;
      T     #BytesListaEventos;

      CALL  "FC897_Generar_PointerAny"
      ( TYP           := 16#10,
        DataTyp       := 16#02,
        repeatcounter := #BytesListaEventos,  // Tamaño del mensaje
        DB_Number     := "JDT2_NDB_UltimoRec",  // DB UltimoRecibido
        storearea     := 16#84,
        storeaddresse := #IniListaEventos,
        Any_Pointer   := #POrigen
      );  // Puntero Origen

      CALL  "FC897_Generar_PointerAny"
      ( TYP           := 16#10,
        DataTyp       := 16#02,
        repeatcounter := #BytesListaEventos,  // Tamaño del mensaje
        DB_Number     := "JDT2_NDB_EventosRec",  // DB EventosRecibidos
        storearea     := 16#84,
        storeaddresse := 16#0000_0000,
        Any_Pointer   := #PDestino
      );  //Puntero Destino

      CALL  BLKMOV
      ( SRCBLK  := #POrigen,
        RET_VAL := #ReturnValor,
        DSTBLK  := #PDestino
      );  // Realizo la transferencia

      JU    MensajeRecibido_OK;



NETWORK
TITLE = Envio del Mensaje ACKN - Acuse de Recibo
// Confirmacion del Mensaje Recibido: Lista de Eventos
// -
// --------------------------------------------------------------------------------------------
// 1º Paso - Guardamos el ID del Mensaje Tratado

MensajeRecibido_OK:NOP   0;

      L     #IDMensaje;  // Guardo el ID del Mensaje Tratado
      T     "DB701_JDT02StatusCOM".ID_UltimoRecibido;

// --------------------------------------------------------------------------------------------
// 2º Paso - Formatear el Mensaje AK en e DB MensajeAK
//    - Rellenar Cabecera
//    - Rellenar Cuerpo

// Rellenar el Campo del ID del Mensaje

      CALL  "FC891_EtiqDInt_EtiqChar"
      ( DB_String   := "JDT2_NDB_AKEmi",  // DB EmisionAK
        Long_String := 4,
        Offset_Ini  := 4,
        Valor       := #IDMensaje
      );

// Preparamos Puntero DB EmisionAK
      L     0;
      LAR1;

// Rellenamos la cabecera del mensaje
      OPN   DB [#DBEmiAK];
      L     2;  // Primer Byte 0x02 - Para que sea enviada
      T     DBB [AR1, P#0.0];
      L     ';';  // Separador
      T     DBB [AR1, P#5.0];

      L     #IdentEmisor;  // Rellenar el Campo Emisor
      T     DBD [AR1, P#6.0];

      L     ';';  // Separador
      T     DBB [AR1, P#10.0];

      L     #IdentReceptor;  // Rellenar el Campo Receptor
      T     DBD [AR1, P#11.0];

      L     ';';  // Separador
      T     DBB [AR1, P#15.0];
      L     '0';  // Tamaño del Mensaje 38
      T     DBB [AR1, P#16.0];
      L     '0038';
      T     DBD [AR1, P#17.0];
      L     ';';  // Separador
      T     DBB [AR1, P#21.0];

// Rellenamos el Evento a escribir- ({ACKN[RSLT]0})
      L     '({';  // Empieza Evento
      T     DBW [AR1, P#22.0];
      L     'ACKN';  // Evento ACKN
      T     DBD [AR1, P#24.0];

      L     '[';  // Atributo del Evento RSLT
      T     DBB [AR1, P#28.0];
      L     'RSLT';  // Atributo del Evento RSLT
      T     DBD [AR1, P#29.0];
      L     ']';  // Atributo del Evento RSLT
      T     DBB [AR1, P#33.0];

      L     '0';  // Contestacion del Atributo del Evento AK
      T     DBB [AR1, P#34.0];
      L     '})';  // Final del Evento
      T     DBW [AR1, P#35.0];

// Rellenamos el final del Evento
      L     3;  // Final del Mensaje 0x03
      T     DBB [AR1, P#37.0];

// --------------------------------------------------------------------------------------------
// 3º Paso - Resetear variable para el Timer de Keep Alive
//         - Borrar Mensaje tratado

      SET;
      R     "DB701_JDT02StatusCOM".KeepAlive_Recibido;  // Reseteamos el Timer de KeepAlive

      CALL  "FC898_BorrarMensaje"
      ( DB_A_RESET := "DB704_JDT02UltimoRecibido"  // ¿HAy que borrar asi?
      );  // Damos por acabado el mensaje recibido

      JU    Final;


NETWORK
TITLE = Error del Mensaje, Mal formateado
// - Se da por tratado el mensaje, borrar
//-----------------------------------------------------------------------------------------------
// Error de mensaje, mal formateado

ErrorDeMensajeRecibido:NOP   0;

      CALL  "FC898_BorrarMensaje"
      ( DB_A_RESET := "DB704_JDT02UltimoRecibido"  // ¿Hay que Borrar todo?
      );  // Damos por acabado el Mensaje Recibido

      JU    Final;

NETWORK
TITLE = Finalizar
// Se Acabo la funcion
// - Control del temporizador KA (Reseteo)
// - Volver a Activar el temporizador KA

Final:NOP   0;

//-----------------------------------------------------------------------------------------------
// Paso 1º- Control del temporizador KA

      L     "JDT2_TMPEsperaKA";
      T     #TMPEsperaKA;
      CALL  "FC899_TMP"
      ( Temporizar     := "DB701_JDT02StatusCOM".KeepAlive_Recibido,
        Valor_Tiempo   := #TMPEsperaKA,  // TMP Espera de Recepción de KA
        Base_tiempo_ms := 1000,
        Tiempo_OK      := "DB701_JDT02StatusCOM".TMPEsperaKA_OK,
        Valor_Actual   := "DB701_JDT02StatusCOM".TMPEsperaKA  // Tiempo de 2M
      );

//-----------------------------------------------------------------------------------------------
// Paso 2º - Volver el Temporizador KA, Variable KeepAlive_Recibido = 1

      AN    "DB701_JDT02StatusCOM".KeepAlive_Recibido;
      S     "DB701_JDT02StatusCOM".KeepAlive_Recibido;

END_FUNCTION

FUNCTION "FC703_JDT02EmiJdTMensaje" : Void   // FC703, LAD
TITLE = "EmiJdTMensaje" - Emision de Mensajes
{ S7_Optimized_Access := 'FALSE' }
AUTHOR : TRACKING
NAME : 20141014
VERSION : 4.0
// - Inicializaciones
// - Distrubucion
// - Recoger el Mensaje ACKN
// - Recoger el Mensaje PING o Lista de Eventos
// - Emision del Mensaje
// stored: AutoNumber false, SetENOAutomatically false
   VAR_TEMP
      DBEmiJdT : Word;   // Num. DB de Emision al JdT
      DBUltimoEmi : Word;   // Num. DB del Ultimo Mensaje a Emitir
      DBEmiAK : Word;   // Num. DB del Mensaje AK a Emitir
      Longitud : UDInt;   // Longitud del Mensaje
      CantidadBytes : UDInt;   // Cantidad de Bytes del Mensaje a Enviar
      ReturnValor : Int;   // Temporal
      POrigen : Any;   // Puntero para transferencias y emision
      PDestino : Any;   // Puntero para transferencias
   END_VAR
BEGIN

NETWORK
TITLE = Inicializaciones
// - Inicializa las variables de los DB's
// - Comprueba que el enlace esta activo "EnlaceCP_OK"
// -------------------------------------------------------------------------------------------
// Si trabaja sin Agencia  2018 01 24
      SET;
      AN    "Activar_JDT02";  // Mirar si se trabaja con agencia
      JC    Final;

// ------------------------------------------------------------------------------------------
// Inicializa las variables de los DB's

      L     "JDT2_NDB_EmiMensaje";  // Cogemos el Numero del DB de EmisionMensaje
      T     #DBEmiJdT;
      L     "JDT2_NDB_UltimoEmi";  // Cogemos el Numero del DB de UltimaEmision
      T     #DBUltimoEmi;
      L     "JDT2_NDB_AKEmi";  // Cogemos el Numero del DB de EmisionAK
      T     #DBEmiAK;

// ------------------------------------------------------------------------------------------
// Comprueba el Enlace esta correcto

      A     "DB701_JDT02StatusCOM".EnlaceCP_OK;  // Mirar Si esta el EnlaceCP Activo
      JC    ExisteConexion;  // El EnlaceCP esta OK

// Reseteamos las variables porque El enlaceCP NOK

      R     "DB891_VariablesTCP".TSEND_JdT_PLC_Req_JDT02;  // Resetear Variables
      R     "DB891_VariablesTCP".TSEND_JdT_PLC_Done_JDT02;
      R     "DB891_VariablesTCP".TSEND_JdT_PLC_Error_JDT02;
      R     "DB891_VariablesTCP".TSEND_JdT_PLC_Busy_JDT02;


      JU    Final;  // Finalizar


NETWORK
TITLE = Distribución
// Hay que seguir este orden:
// - Hay que emitir mensaje
// - Hay que recoger el mensaje ACKN
// - Hay que recoger el mensaje PING o Lista de Eventos
ExisteConexion:NOP   0;

// ------------------------------------------------------------------------------------------
// Hay que emitir mensaje

      L     0;  // Ya tenemos mensaje a Emitir
      LAR1;
      OPN   DB [#DBEmiJdT];
      L     DBB [AR1, P#0.0];
      L     0;
      <>I;
      JC    EmitirMensaje;  // Ir a Emitir

// ------------------------------------------------------------------------------------------
// Hay que recoger Mensaje ACKN para emitir

      L     0;
      LAR1;
      OPN   DB [#DBEmiAK];
      L     DBB [AR1, P#0.0];
      L     2;
      ==I;
      JC    EmitirEvento_AcuseRecibo;  // Ir a Recoger el mensaje AK

// ------------------------------------------------------------------------------------------
// Hay que recoger Mensaje PING o Lista de Eventos para Emitir

      L     0;
      LAR1;
      OPN   DB [#DBUltimoEmi];
      L     DBB [AR1, P#0.0];
      L     2;
      ==I;
      JC    EmitirEvento;  // Ir a Recoger el mensaje KA o de Eventos

      JU    Final;



NETWORK
TITLE = Recoger el Mensaje ACKN - Confirmacion
// Pasos a Seguir:
// - Calcular la Longitud del Mensaje (Puede ser variable)
// - Generamos los punteros Origen y Destino
// - Transferir el Mensaje para Emitir
// - Borrar el Mensaje AK, para decir que lo hemos tratado, y Resetear Variables
// - Emitimos el Mensaje
EmitirEvento_AcuseRecibo:NOP   0;

// ------------------------------------------------------------------------------------------
// 1º Paso - Calcular la longitud del Mensaje

      CALL  "FC890_EtiqChar_EtiqDInt"
      ( DB_String   := "JDT2_NDB_AKEmi",
        Long_String := 5,
        Offset_Ini  := 20,
        Valor       := #Longitud
      );

      L     #Longitud;
      T     #CantidadBytes;

// ------------------------------------------------------------------------------------------
// 2º Paso - Generamos los punteros Origen y Destino

      CALL  "FC897_Generar_PointerAny"
      ( TYP           := 16#10,
        DataTyp       := 16#02,
        repeatcounter := #CantidadBytes,  // Tamaño del mensaje
        DB_Number     := "JDT2_NDB_AKEmi",  // DB donde esta guardado el EmisionAK
        storearea     := 16#84,
        storeaddresse := 16#0000_0000,
        Any_Pointer   := #POrigen  // Puntero del EmisionAK
      );

      CALL  "FC897_Generar_PointerAny"
      ( TYP           := 16#10,
        DataTyp       := 16#02,
        repeatcounter := #CantidadBytes,  // Tamaño del mensaje
        DB_Number     := "JDT2_NDB_EmiMensaje",  // DB donde guardar el EmisionMensaje
        storearea     := 16#84,
        storeaddresse := 16#0000_0000,
        Any_Pointer   := #PDestino  // Puntero del Mensaje a Enviar
      );

// ------------------------------------------------------------------------------------------
// 3º Paso - Transferir en Mensaje para emitir

      CALL  BLKMOV
      ( SRCBLK  := #POrigen,
        RET_VAL := #ReturnValor,
        DSTBLK  := #PDestino
      );

// ------------------------------------------------------------------------------------------
// 4º Paso - Borrar el Mensaje AK y Resetear variables internas

      CALL  "FC898_BorrarMensaje"
      ( DB_A_RESET := "DB706_JDT02EmisionAK"  // ¿Hay que borrar asi?
      );  // Damos por acabado el envio del mensaje

      SET;  // Ya hay Actividad
      R     "DB701_JDT02StatusCOM".SinActividad;

// ------------------------------------------------------------------------------------------
// 5º Paso - Pasamos a Emitir el Mensaje

      L     #CantidadBytes;
      T     "DB701_JDT02StatusCOM".EmiJdT_Longitud;  // Guardamos la longitud para la Emision
      JU    EmitirMensaje;



NETWORK
TITLE = Recoger el Mensaje KA o Lista de Eventos
// Pasos a Seguir:
// - Calcular la Longitud del Mensaje(Puede ser variable)
// - Generamos los punteros Origen y Destino
// - Transferir el Mensaje para Emitir
// - Borrar el Mensaje AK, para decir que lo hemos tratado, y Resetear Variables
// - Emitimos el Mensaje
EmitirEvento:NOP   0;

// ------------------------------------------------------------------------------------------
// 1º Paso - Calcular la longitud del Mensaje

      CALL  "FC890_EtiqChar_EtiqDInt"
      ( DB_String   := "JDT2_NDB_UltimoEmi",
        Long_String := 5,
        Offset_Ini  := 20,
        Valor       := #Longitud
      );

      L     #Longitud;
      T     #CantidadBytes;

// ------------------------------------------------------------------------------------------
// 2º Paso - Generamos los punteros Origen y Destino

      CALL  "FC897_Generar_PointerAny"
      ( TYP           := 16#10,
        DataTyp       := 16#02,
        repeatcounter := #CantidadBytes,  // Tamaño del mensaje
        DB_Number     := "JDT2_NDB_UltimoEmi",  // DB donde esta guardado el UltimoMensaje
        storearea     := 16#84,
        storeaddresse := 16#0000_0000,
        Any_Pointer   := #POrigen  // Puntero del UltimoMensaje
      );

      CALL  "FC897_Generar_PointerAny"
      ( TYP           := 16#10,
        DataTyp       := 16#02,
        repeatcounter := #CantidadBytes,  // Tamaño del mensaje
        DB_Number     := "JDT2_NDB_EmiMensaje",  // DB donde guardar el Emisio del Mensaje
        storearea     := 16#84,
        storeaddresse := 16#0000_0000,
        Any_Pointer   := #PDestino  // Puntero del Mensaje a Enviar
      );

// ------------------------------------------------------------------------------------------
// 3º Paso - Transferir

      CALL  BLKMOV
      ( SRCBLK  := #POrigen,
        RET_VAL := #ReturnValor,
        DSTBLK  := #PDestino
      );

// ------------------------------------------------------------------------------------------
// 4º Paso - Borrar el Mensaje Tratado y Resetear variables internas

      SET;  // Ya hay Actividad
      R     "DB701_JDT02StatusCOM".SinActividad;

// Parar Borrar el Mensaje hay que saber de que tipo es:
// KA o Lista de Eventos - Porque se hace cosas diferentes

      L     0;
      LAR1;
      OPN   DB [#DBUltimoEmi];
      L     DBD [AR1, P#24.0];
      L     'PING';
      <>I;
      JC    _040;  // Si no es KA hay que borrarlo entero

// Es Mensaje KA - Borrar todo el Mensaje
      CALL  "FC898_BorrarMensaje"
      ( DB_A_RESET := "DB705_JDT02UltimoEnviado"  // ¿Hay que borrar asi?
      );  // Damos por acabado el envio del mensaje KA

      JU    _041;

// Es Mnesaje de Lista de Eventos lo damos por tratado
_040: OPN   DB [#DBUltimoEmi];  // Damos por enviado el mensaje de Evento
      L     'N';
      T     DBB [AR1, P#0.0];

      JU    _041;

// ------------------------------------------------------------------------------------------
// 5º Paso - Pasamos a Emitir el Mensaje

_041: L     #CantidadBytes;
      T     "DB701_JDT02StatusCOM".EmiJdT_Longitud;  // Guardamos la longitud para la Emision
      JU    EmitirMensaje;



NETWORK
TITLE = Emision del Mensaje
// Pasos a Seguir
// - Control de la Emision
// - Calcular el puntero de lo que tenemos que emitir
// - Emision del Mensaje
// - Comprobacion del Mensaje Enviado
EmitirMensaje:NOP   0;

// ------------------------------------------------------------------------------------------
// 1º Paso - Control de la Emision

      AN    "DB891_VariablesTCP".TSEND_JdT_PLC_Busy_JDT02;
      AN    "DB891_VariablesTCP".TSEND_JdT_PLC_Req_JDT02;
      AN    "DB891_VariablesTCP".TSEND_JdT_PLC_Flanco_JDT02;
      =     "DB891_VariablesTCP".TSEND_JdT_PLC_Flanco_JDT02;

      A     "DB891_VariablesTCP".TSEND_JdT_PLC_Flanco_JDT02;
      AN    "DB891_VariablesTCP".TSEND_JdT_PLC_Req_JDT02;
      S     "DB891_VariablesTCP".TSEND_JdT_PLC_Req_JDT02;


// ------------------------------------------------------------------------------------------
// 2º Paso - Generar el Puntero de lo que se tiene que Emitir

      CALL  "FC897_Generar_PointerAny"
      ( TYP           := 16#10,
        DataTyp       := 16#02,
        repeatcounter := "DB701_JDT02StatusCOM".EmiJdT_Longitud,  // Tamaño del mensaje
        DB_Number     := "JDT2_NDB_EmiMensaje",  // DB donde esta guardado el EmisionMensaje
        storearea     := 16#84,
        storeaddresse := 16#0000_0000,
        Any_Pointer   := #POrigen  // Puntero del EmisionMensaje
      );

// ------------------------------------------------------------------------------------------
// 2º Paso - Emision del Mensaje

      CALL  TSEND, "DB898_TSEND_JdT_PLC_JDT02"
      ( REQ    := "DB891_VariablesTCP".TSEND_JdT_PLC_Flanco_JDT02,
        ID     := W#16#3,
        LEN    := "DB701_JDT02StatusCOM".EmiJdT_Longitud,
        DONE   := "DB891_VariablesTCP".TSEND_JdT_PLC_Done_JDT02,
        BUSY   := "DB891_VariablesTCP".TSEND_JdT_PLC_Busy_JDT02,
        ERROR  := "DB891_VariablesTCP".TSEND_JdT_PLC_Error_JDT02,
        STATUS := "DB891_VariablesTCP".TSEND_JdT_PLC_Status_JDT02,
        DATA   := #POrigen
      );



// ------------------------------------------------------------------------------------------
// 3º Paso - Comprobacion del Mensaje Enviado

      A     "DB891_VariablesTCP".TSEND_JdT_PLC_Req_JDT02;  // Si llega Error en la Emision
      AN    "DB891_VariablesTCP".TSEND_JdT_PLC_Done_JDT02;  // Restear
      A     "DB891_VariablesTCP".TSEND_JdT_PLC_Error_JDT02;
      S     "DB701_JDT02StatusCOM".EmiJdT_Reset;
      R     "DB891_VariablesTCP".TSEND_JdT_PLC_Req_JDT02;

      A     "DB891_VariablesTCP".TSEND_JdT_PLC_Req_JDT02;  // Si llega que la Emision es OK
      A     "DB891_VariablesTCP".TSEND_JdT_PLC_Done_JDT02;
      AN    "DB891_VariablesTCP".TSEND_JdT_PLC_Error_JDT02;
      R     "DB891_VariablesTCP".TSEND_JdT_PLC_Req_JDT02;

      JCN   NoEmitidoMensaje;

      R     "DB701_JDT02StatusCOM".EmiJdT_PeticionActiva;
      CALL  "FC898_BorrarMensaje"
      ( DB_A_RESET := "DB703_JDT02EmisionMensaje"  // ¿Hay que borralo asi?
      );

NoEmitidoMensaje:JU    Final;


NETWORK
TITLE = Finalizar
// - Finaliza la función
Final:NOP   0;

END_FUNCTION

FUNCTION "FC789_Tratamiento_mensajes_Router" : Void   // FC789, LAD
{ S7_Optimized_Access := 'FALSE' }
// stored: AutoNumber false, SetENOAutomatically false
   VAR_TEMP
      separador : Char;
      final : Char;
      ESPACIO : Char;
      retval_split : Int;
      retval : Int;
      posicion_split : UDInt;
      modo_split : DWord;
      numero_mensajes : Int;
      contador : Int;
      tamaño : Int;
      EVENTO_MENSAJE : String[4];
   END_VAR
   VAR_TEMP   // added for the SCL form of the ladder/FBD networks
      _w1 : Bool;
      _w2 : Bool;
   END_VAR
BEGIN

REGION Network 1 (SCL): inicialización
   REGION inicialiacion
       #final := ' ';
       #separador := ';';
       #modo_split := 0;
       #modo_split.%X0 := false;
       #modo_split.%X1 := true;
       #modo_split.%X3 := FALSE;
       #modo_split.%X4 := true;
       #posicion_split := 0;
       #ESPACIO := ' ';
       #numero_mensajes := 0;

       // evaluo si hay algun mensaje que impida que pueda realizar la segmentación del nuevo bloque
       // 
      #tamaño:= LEN("DB199_eventos_convertidos".evento[0]);

   END_REGION
END_REGION

REGION Network 2
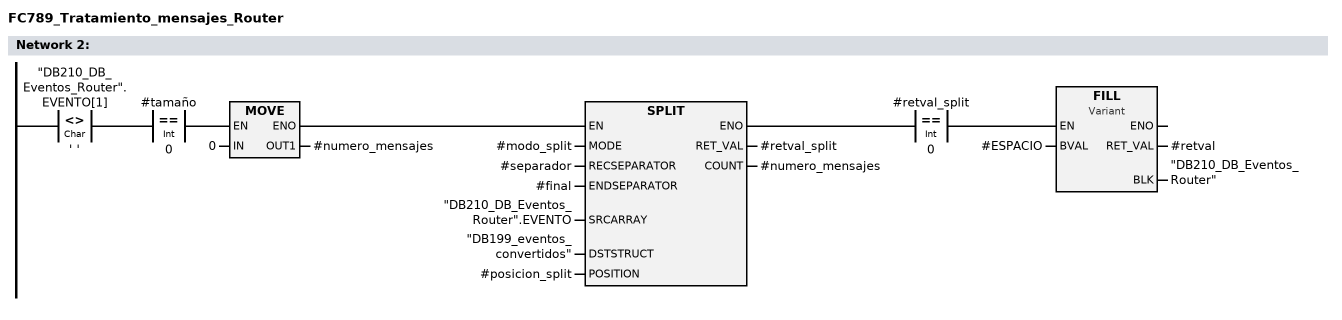
   RUNG wire#powerrail
      { S7_Templates := "SrcType := Char" } NE_Contact(in1 := "DB210_DB_Eventos_Router".EVENTO[1], in2 := ' ')
      { S7_Templates := "SrcType := Int" } EQ_Contact(in1 := #tamaño, in2 := 0)
      Move(in := 0, out1 => #numero_mensajes)
      SPLIT(Mode := #modo_split, RecSeparator := #separador, EndSeparator := #final, SrcArray := "DB210_DB_Eventos_Router".EVENTO, DstStruct := "DB199_eventos_convertidos", Position := #posicion_split, Ret_Val => #retval_split, Count => #numero_mensajes)
      { S7_Templates := "SrcType := Int" } EQ_Contact(in1 := #retval_split, in2 := 0)
      { S7_Templates := "ptr_type := Variant" } FILL(BVAL := #ESPACIO, RET_VAL => #retval, BLK => "DB210_DB_Eventos_Router")
   END_RUNG
   // the same network as SCL:
   #_w1 := ("DB210_DB_Eventos_Router".EVENTO[1] <> ' ') AND (#tamaño = 0);
   IF #_w1 THEN #numero_mensajes := 0; END_IF;
   #retval_split := SPLIT(EN := #_w1,
                          Mode := #modo_split,
                          RecSeparator := #separador,
                          EndSeparator := #final,
                          SrcArray := "DB210_DB_Eventos_Router".EVENTO,
                          DstStruct := "DB199_eventos_convertidos",
                          Position := #posicion_split,
                          Count => #numero_mensajes,
                          ENO => #_w2);
   IF #_w2 AND (#retval_split = 0) THEN
       #retval := FILL(BVAL := #ESPACIO, BLK => "DB210_DB_Eventos_Router");
   END_IF;
END_REGION

REGION Network 3 (SCL): Bucle que recorre mensajes
   IF #numero_mensajes>0 THEN
       FOR #contador := 0 TO #numero_mensajes  BY 1 DO

           // voy a tener en cuenta que los cuatro primeros caracteres del string convertido siempre van a ser el tipo de mensaje que tengo que tratar
           // 
           #EVENTO_MENSAJE := LEFT(IN := "DB199_eventos_convertidos".evento[#contador], L := 4);

           REGION Evento_RUES
               IF #EVENTO_MENSAJE = 'RUES' THEN
                   // GENERO UNA RUTA DE ELTIQUETA ESPECIAL
                   "FC782_Evento_RUES"(#contador);
                   "DB199_eventos_convertidos".evento[#contador] := DELETE(IN := "DB199_eventos_convertidos".evento[#contador], L := 0, P := 0);
                   #numero_mensajes -= 1;
                   CONTINUE;
               END_IF;
           END_REGION

           REGION Evento_RUET
               IF #EVENTO_MENSAJE = 'RUET' THEN
                   "FC780_Evento_RUET"(#contador);

                   "DB199_eventos_convertidos".evento[#contador] := DELETE(IN := "DB199_eventos_convertidos".evento[#contador], L := 0, P := 0);
                   #numero_mensajes -= 1;
                   CONTINUE;
           END_IF;
           END_REGION

           REGION Evento_BOET
               IF #EVENTO_MENSAJE = 'BOET' THEN
                   // ELIMINO UNA ETIQUETA DE LA BBDD

                   "FC783_Evento_BOET"(#contador);
                   "DB199_eventos_convertidos".evento[#contador] := DELETE(IN := "DB199_eventos_convertidos".evento[#contador], L := 0, P := 0);
                   #numero_mensajes -= 1;
                   CONTINUE;
               END_IF;
           END_REGION

           REGION Evento_BOBD
               IF #EVENTO_MENSAJE = 'BOBD' THEN
                   // BORRO LA BBDD   
                   "FC900_Reset_DB_Offset"(DB_A_RESET := "DB212_Cola_Activa",
                                           BORRAR_DESTE_BYTE := 0);
                   "FC900_Reset_DB_Offset"(DB_A_RESET := "DB201_RegEtiquetas_0001_1000",
                                           BORRAR_DESTE_BYTE := 0);
                   "FC900_Reset_DB_Offset"(DB_A_RESET := "DB202_RegEtiquetas_1001_2000",
                                           BORRAR_DESTE_BYTE := 0);
                   "FC900_Reset_DB_Offset"(DB_A_RESET := "DB203_RegEtiquetas_2001_3000",
                                           BORRAR_DESTE_BYTE := 0);
                   "FC900_Reset_DB_Offset"(DB_A_RESET := "DB204_RegEtiquetas_3001_4000",
                                           BORRAR_DESTE_BYTE := 0);
                   "FC900_Reset_DB_Offset"(DB_A_RESET := "DB209_Reg_Etquetas_Esp_Activa",
                                           BORRAR_DESTE_BYTE := 0);
                   // supervisión de los mensajes tratados. borrar luego
                   // 

                   // borrado del evento que ya hemos tratado
                   "DB199_eventos_convertidos".evento[#contador] := DELETE(IN := "DB199_eventos_convertidos".evento[#contador], L := 0, P := 0);
                   #numero_mensajes -= 1;
                   CONTINUE;
               END_IF;
           END_REGION
           REGION Evento_ORDE
               IF #EVENTO_MENSAJE = 'ORDE' THEN
                   // MENSAJE ORDE EN MESA

                   "FC781_Evento_ORDE"(#contador);
                   "DB199_eventos_convertidos".evento[#contador] := DELETE(IN := "DB199_eventos_convertidos".evento[#contador], L := 0, P := 0);
                   #numero_mensajes -= 1;
                   CONTINUE;
               END_IF;
           END_REGION
           REGION Evento_INIR
               IF #EVENTO_MENSAJE = 'INIR' THEN
                   //MENSAJE DE INCIALIZACION

                   "FC784_Evento_INIR"(#contador);
                   "DB199_eventos_convertidos".evento[#contador] := DELETE(IN := "DB199_eventos_convertidos".evento[#contador], L := 0, P := 0);
                   #numero_mensajes -= 1;
                   CONTINUE;
               END_IF;
           END_REGION

           // Statement section FOR

       END_FOR;

   END_IF;
END_REGION
END_FUNCTION

FUNCTION "FC519_Buc_Lec_Scanners" : Void   // FC519, STL
{ S7_Optimized_Access := 'FALSE' }
AUTHOR : SSCC
NAME : 23062013
VERSION : 3.2
// stored: AutoNumber false
   VAR_TEMP
      NDB_TMP : Word;   // Num. DB Temporal
      PunteroTMP : DWord;   // Puntero Temporal
      DBNodosPresentes : UInt;   // DB De Nodos Presentes de la Red
      RedActual : UInt;   // Red actual de Lectura
      SCR_Actual : UInt;
      CNT_LectCiclo : UInt;   // Contador de lecturas en la Red
   END_VAR
BEGIN

NETWORK
TITLE = Inicializaciones
// --------------------------------------------------------------------------------------
// --- Incializar para recorrer las Redes de Escanneres

      L     1;
      T     #RedActual;



NETWORK
TITLE = Bucle de scanners
// --------------------------------------------------------------------------------------
// --- Inicializar datos de la Red de Scanners

_INI: NOP   0;

// --------------------------------------------------------------------------------------
// --- Comprobar si está configurada

      L     "DB911_Conf_Sistema_Scanners".Bucles_lectura_Scanner[#RedActual].NodoInicial;  // Si el Nodo Incial es cero
      L     0;  // No existe Scanner en la Red
      ==I;
      JC    _FIN;

// --------------------------------------------------------------------------------------
// --------------------------------------------------------------------------------------
// --- Lecturas de los Escaneres de la Red  (Bucle)

// --------------------------------------------------------------------------------------
// --- Incializaciones del Bucle

      L     0;  // --- Inicio Contador lecturas tradadas por ciclo
      T     #CNT_LectCiclo;

// --------------------------------------------------------------------------------------
// --- Comprobaciones del Nodo Actual a Comprobar

      L     "DB911_Conf_Sistema_Scanners".Bucles_lectura_Scanner[#RedActual].SCR_Actual;  // --- Comparamos con el numero de Scanneres definidos
      L     "DB911_Conf_Sistema_Scanners".Bucles_lectura_Scanner[#RedActual].NodoInicial;  //     Si estamos dentro de la Red de Scanners
      >=I;
      JC    ISRC;

      L     "DB911_Conf_Sistema_Scanners".Bucles_lectura_Scanner[#RedActual].NodoInicial;
      T     "DB911_Conf_Sistema_Scanners".Bucles_lectura_Scanner[#RedActual].SCR_Actual;  // --- Inicimos el Número de Scanner a tratar de 0..n

ISRC: L     "DB911_Conf_Sistema_Scanners".Bucles_lectura_Scanner[#RedActual].SCR_Actual;
      L     "DB911_Conf_Sistema_Scanners".Bucles_lectura_Scanner[#RedActual].NodoFinal;  // --- Comparamos con el numero de Scanners definidos
      <=I;  //     Si estamos en el ultimo ponemos al Inicio de la Red.
      JC    TIPO;  //    SPB   BSRC

      L     "DB911_Conf_Sistema_Scanners".Bucles_lectura_Scanner[#RedActual].NodoInicial;
      T     "DB911_Conf_Sistema_Scanners".Bucles_lectura_Scanner[#RedActual].SCR_Actual;  // --- Inicimos el Número de Scanner a tratar de 0..n


TIPO: SET;  // Comprobamos si es nodo profibus o profinet para hacer el diagnóstico dentro de la red
// -- si estamos en modo simulacion no hacemos ningún diagnostico de nodo
      SET;
      A     "Activar_Simulador";
      JC    comprobar_si_hay_etiqueta;

// -- Comprobamos el tipo de modelo para hacer el diagnostico del nodo
      L     "DB911_Conf_Sistema_Scanners".Bucles_lectura_Scanner[#RedActual].Modelo;
      L     DINT#5;
      >=I;
      JC    bucle_profinet;  // bucle de profinet



NETWORK
TITLE = Comprobacion de Nodos
//*******************************************************************************
// --- Comprobacion si el Nodo existe   (ZONA PROFIBUS)
// ZONA DE PROFIBUS QUEDA COMENTADA POR ESTAR CASI OBSOLETA
// DE QUERER ACTIVARLA OTRA VEZ, DESCOMENTAR LA ZONA MARCADA ENTRE INICIO Y FIN
//-- INICIO ZONA PROFIBUS 20200508

      L     #DBNodosPresentes;  // --- Formatea DB Errores Para poder Abrirlo
      T     #NDB_TMP;

      L     P#52.0;  // --- Direccion del Bit dentro del DB de Errores
      L     "DB911_Conf_Sistema_Scanners".Bucles_lectura_Scanner[#RedActual].SCR_Actual;  //     Bit del Nodo Presente (Actual)
      +D;
      L     1;
      -D;
      T     #PunteroTMP;

      OPN   DB [#NDB_TMP];  // --- Existe Nodo ?
      SET;
      A     DBX [#PunteroTMP];
      JC    Siguiente_Scanner;

      L     #PunteroTMP;  // --- Direccion del Bit dentro del DB de Errores
      L     128;  //     Bit del Error del Nodo (Actual)
      +D;
      T     #PunteroTMP;

      OPN   DB [#NDB_TMP];  // --- Nodo en Error ?
      SET;
      A     DBX [#PunteroTMP];
      JC    Siguiente_Scanner;

      JU    comprobar_si_hay_etiqueta;  // salta a la comprobación

//-- FIN ZONA PROFIBUS 20200508
//*******************************************************************************


//================================================================================
// --- Comprobacion si el Nodo existe   (ZONA PROFINET)
bucle_profinet:SET;

      L     "DB911_Conf_Sistema_Scanners".Bucles_lectura_Scanner[#RedActual].SCR_Actual;
      T     #SCR_Actual;

      SET;
      AN    "DB927_PNIODiag_Data".RED[1].NODO[#SCR_Actual].OK;
      JC    Siguiente_Scanner;

//================================================================================


NETWORK
TITLE = Comprobación de si existe etiqueta
// ------------------------------------------------------------------------------
// --- Mirar y Extraer la Eiqueta del Nodo Actual del Scanner
// --- Llamada a la lectura dependiendo de Modelo

comprobar_si_hay_etiqueta:NOP   0;



      L     "DB911_Conf_Sistema_Scanners".Bucles_lectura_Scanner[#RedActual].Modelo;  // --- Reparto por Modelo de Scanner
      JL    LSTX;

      JU    DATL;  // --- Modelo DataLogic profibus  (0)
      JU    SICK;  // --- Modelo SICK profibus      (1)
      JU    SICA;  // --- Modelo SICK para router alfanumérico  profibus  (2)
      JU    Siguiente_Scanner;  // --- RESERVA PROFIBUS
      JU    Siguiente_Scanner;  // --- RESERVA PROFIBUS
      JU    SICN;  // --- Modelo SICK para profinet (5) Añadido Nieves 17/08/16
      JU    SIAN;  // --- Modelo SICK ALFANUMERICO para profinet (6) Añadido Nieves 17/08/16
      JU    SILINT;  // MODELO SICK PARA ETIQUETAS ULINT (7)

LSTX: JU    Siguiente_Scanner;  // --- No definido


// ------------------------------------------------------------------------------
// --- Tratamiento de Scanner de Modelo DataLogic profibus

DATL: NOP   0;
//      CALL  "FC524_Form_Lec_Modelo_DL"
//         Red_Actual    :=#RedActual
//         Datos_Red     :=#Datos_Red
//         CNT_LectCiclo :=#CNT_LectCiclo

// en caso de que sea necesario recuperar la función,
// recoger de librería obsoletos scanners
      JU    Siguiente_Scanner;

// ------------------------------------------------------------------------------
// --- Tratamiento de Scanner de Modelo SICK profibus

SICK: NOP   0;
//  CALL  "FC525_Form_Lect_Modelo_SICK"
//         Red_Actual    :=#RedActual
//         Datos_Red     :=#Datos_Red
//         CNT_LectCiclo :=#CNT_LectCiclo

// en caso de que sea necesario recuperar la función,
// recoger de librería obsoletos scanners

      JU    Siguiente_Scanner;


// ------------------------------------------------------------------------------
// --- Tratamiento de Scanner de Modelo SICK para router alfanumérico profibus

SICA: NOP   0;

//   CALL  "FC526_Form_Lec_Modelo_SICK_ALF"
//         Red_Actual    :=#RedActual
//         Datos_Red     :=#Datos_Red
//         CNT_LectCiclo :=#CNT_LectCiclo

// en caso de que sea necesario recuperar la función,
// recoger de librería obsoletos scanners

      JU    Siguiente_Scanner;

// ------------------------------------------------------------------------------
// --- Tratamiento de Scanner de Modelo SICK profinet

SICN: SET;
      CALL  "FC527_Form_Lec_Modelo_SICK_PN"
      ( Numero_Red    := #RedActual,
        Datos_red     := "DB911_Conf_Sistema_Scanners".Bucles_lectura_Scanner[#RedActual],
        CNT_LectCiclo := #CNT_LectCiclo
      );

      JU    Siguiente_Scanner;


// ------------------------------------------------------------------------------
// --- Tratamiento de Scanner de Modelo SICK para router alfanumérico profinet


SIAN: SET;
      CALL  "FC528_Form_Lec_Mod_SICK_PN_ALF"
      ( Numero_Red    := #RedActual,
        Datos_Red     := "DB911_Conf_Sistema_Scanners".Bucles_lectura_Scanner[#RedActual],
        CNT_LectCiclo := #CNT_LectCiclo
      );


SILINT:SET;
      CALL  "FC529_Form_Lec_Modelo_SICK_PN_ULINT"
      ( Numero_Red    := #RedActual,
        Datos_red     := "DB911_Conf_Sistema_Scanners".Bucles_lectura_Scanner[#RedActual],
        CNT_LectCiclo := #CNT_LectCiclo
      );

      JU    Siguiente_Scanner;

// ------------------------------------------------------------------------------



NETWORK
TITLE = pasar al siguiente scanner

// ------------------------------------------------------------------------------
// --- Maximas Lecturas de Ciclo en la Red

Siguiente_Scanner:NOP   0;
      L     #CNT_LectCiclo;  // --- Valida la cantidad Maxima de lecturas tratadas por ciclo
      L     "ROUT_Max_Lec_Ciclo";  // L     "DB911_Conf_Sistema_Router".Num_Max_Lec_Ciclo
      >=I;
      JC    FSRC;

// ------------------------------------------------------------------------------------------------
// --- Nodo Siguiente de la Red

      L     1;
      L     "DB911_Conf_Sistema_Scanners".Bucles_lectura_Scanner[#RedActual].SCR_Actual;  // Incrementamos el scanner que debe de ser tratado
      +I;
      T     "DB911_Conf_Sistema_Scanners".Bucles_lectura_Scanner[#RedActual].SCR_Actual;

      SET;
      L     "DB911_Conf_Sistema_Scanners".Bucles_lectura_Scanner[#RedActual].SCR_Actual;  // Si estamos en el ultimo salimos del Bucle
      L     "DB911_Conf_Sistema_Scanners".Bucles_lectura_Scanner[#RedActual].NodoFinal;  // Comparamos con el numero de Scanners definidos
      <=I;
      JC    TIPO;  //  SPB   BSRC

// ------------------------------------------------------------------------------------------------
// --- Final del Bucle

FSRC: NOP   0;


// --------------------------------------------------------------------------------------
// --------------------------------------------------------------------------------------
// --------------------------------------------------------------------------------------
// --------------------------------------------------------------------------------------
// --------------------------------------------------------------------------------------
// --------------------------------------------------------------------------------------



// --------------------------------------------------------------------------------------
// --- Siguiente Red

      L     #RedActual;  // Ultima Red a Testear
      L     5;  // Red --> 1...5
      ==I;
      JC    _FIN;

      L     #RedActual;  // Siguiente Red Scanneres
      L     1;
      +I;
      T     #RedActual;

      JU    _INI;  // A Testear Siguiente Red




NETWORK
TITLE = 
// --------------------------------------------------------------------------------------
// --- Final de la Funcion

_FIN: NOP   0;



END_FUNCTION

FUNCTION "FC528_Form_Lec_Mod_SICK_PN_ALF" : Void   // FC528, STL
{ S7_Optimized_Access := 'FALSE' }
AUTHOR : ROUTER_A
NAME : 20181011
VERSION : 3.4
// stored: AutoNumber false
   VAR_INPUT
      Numero_Red : UInt;   // Red Actual de Lectura
      Datos_Red : "ROUT_Conf_Bucle_Lect_SCR";
   END_VAR
   VAR_IN_OUT
      CNT_LectCiclo : UInt;
   END_VAR
   VAR_TEMP
      Datos_E_Scanner : Array[0.."ROUT_Long_Dat_Scanner"] of Byte;
      EAB_Lectura : UInt;   // Byte 0 Entradas/Salidas del Scanner
      Datos_Diagnostico : Word;
      PunteroSCR_A : DWord;
      caracter_relleno : Char;
      retvalue : Int;
      Numero_Caracteres : UInt;
      CNT_Escritura : UInt;
      SCR_Actual : UInt;
      NumScanner : UInt;
      AUX_NumScanner : UInt;
      cero : Byte;
      CNT_Lectura : UInt;
      CNT_Datos_Pantalla : UInt;
   END_VAR
BEGIN

NETWORK
TITLE = Inicializar
// -- Calcular la dirección de lectura del scanner actual

      L     #Datos_Red.SCR_Actual;  // Direccion de E/S de Scanner
      L     #Datos_Red.NodoInicial;  // (Nodo * Long. Datos) + Address Incio
      -I;
      L     "ROUT_Long_Dat_Scanner";
      *I;
      L     #Datos_Red.AddresInicial;
      +I;
      T     #EAB_Lectura;

      L     0;
      T     #cero;


// ----------------------------------------------------------------------
// --- Calculo de Punteros   E / S

      L     #EAB_Lectura;  //--- Obtener Direccion entrada Scanner
      SLD   3;  //    Dar formato de Integer a Puntero
      L     P#3.0;  //--  EB_Lectura + 3 Byte
      +D;  //    Leer de PAB
      T     #PunteroSCR_A;

// -------------------------------------------------------------------------------------
// --- Numero de SCR Actual

      L     #Datos_Red.SCR_Actual;
      T     #SCR_Actual;


// -------------------------------------------------------------------------------------

// -------------------------------------------------------------------------------------
// obtener el caracter de relleno

      L     "ROUT_CaracterRelleno";
      T     #caracter_relleno;
// -------------------------------------------------------------------------------------


NETWORK
TITLE = Determinar Nueva Lectura
// -------------------------------------------------------------------------------------
// recogida de todos los datos del scanner

      CALL  "FC570_Leer_Zona_Entradas"
      ( Inicio_Zona := #EAB_Lectura,
        Long_Zona   := "ROUT_Long_Dat_Scanner",
        Datos_Zona  := #Datos_E_Scanner
      );

// Nieves: hay que revisar en un funcionamiento con scanner real
//  como quedan los datos de diagnóstico


      L     #Datos_E_Scanner[0];
      T     #Datos_Diagnostico.%B0;
      L     #Datos_E_Scanner[1];
      T     #Datos_Diagnostico.%B1;


// -------------------------------------------------------------------------------------
// ---  pasamos a ver el telegrama del scanner
// --- Comprobamos si hay Nueva Lectura de Scanner
// --- si el número de lectura disponible es igual a la ultima tratada
// --- Significa que no hay ninguna nueva lectura pendiente de ser tratada


      L     "DB214_CNT_Mens_SCR".RedScanners[#Numero_Red].CNT_NODO_PROF_SCR[#SCR_Actual];  // --- Memoria con el número de la ultima lectura tratada
      L     #Datos_E_Scanner[3];  // --- Numero de lectura disponible para ser tratada
      ==I;
      JC    Fin_funcion;

// -------------------------------------------------------------------------------------


NETWORK
TITLE = Obtener Identificador Scanner (modif a 3digit el 27/08/18)

// -------------------------------------------------------------------------------------
// --- Numero de Numero del Scanner
      L     #Datos_E_Scanner[7];  // --- Obtener Centenas
      L     W#16#F;  //     Eliminamos la parte alta del BYTE
      AW;  //     Multiplicamos por el peso del caracter
      L     100;
      *I;
      T     #AUX_NumScanner;  // --- Lo Paso al valor del NODO

      L     #Datos_E_Scanner[8];  // --- Obtener Decenas
      L     W#16#F;  //     Eliminamos la parte alta del BYTE
      AW;  //     Multiplicamos por el peso del caracter
      L     10;
      *I;
      L     #AUX_NumScanner;  // --- Lo sumamo al valor del NODO
      +I;
      T     #AUX_NumScanner;  // --- Lo sumamo al valor del NODO


      L     #Datos_E_Scanner[9];  // --- Obtener Unidad
      L     W#16#F;  //     Eliminamos la parte alta del BYTE
      AW;  //     Multiplicamos por el peso del caracter
      L     1;
      *I;
      L     #AUX_NumScanner;  // --- Lo sumamo al valor del NODO
      +I;
      T     #NumScanner;  // --- Lo sumamo al valor del NODO

// -------------------------------------------------------------------------------------
// -- si el numero del scanner es 0, ha habido algún problema NIEVES PENDIENTE DEFINIR

      SET;
      L     #NumScanner;  // -- Descartar cualquier lectura de identificadores de scanner 0
      L     0;
      ==I;
      JC    Fin_Bucle;

// -------------------------------------------------------------------------------------


NETWORK
TITLE = Validar Escritura en DB e inicar Registros
// -------------------------------------------------------------------------------------
// --- Comprobacion de nuemro de caracteres leidos

      L     "ROUT_Long_Etiqueta";  // --- Carga Dato de Número de caracteres de etiquetas esperados en el DB
      L     4;  // -- le añadimos 4 porque los 4 digitos qu emanda de identificador nos se guardan realmente pero se cuentan en el mensaje.
      +I;
      L     #Datos_E_Scanner[5];  // --- Carga el dato de Número de caracteres Leidos
      -I;
      T     #Numero_Caracteres;  // --- Posición donde empezar a escribir la etiqueta en DB

      SET;
      L     #Numero_Caracteres;
      L     0;
      <=I;
      JC    Error_lectura;  // --- Si resultado <=0 LONGITUD LECTURA de scanner FUERA DE RANGO


// -------------------------------------------------------------------------------------
// --- Validar si se puede leer la nueva lectura
// --- la condición es que la lectura anterior esté tratada

      SET;
      L     "DB211_Lecturas_Scanner".Lec_Scanner[#NumScanner].Lectura_SCR[0];
      L     'N';  //      Carga el caracter 'N' para compara
      ==I;  //      Si es igual no tratamos la lectura actual
      JC    Fin_funcion;  //      ESPERAMOS QUE SE TRATE LA LECTURA ANTERIOR

// -------------------------------------------------------------------------------------


NETWORK
TITLE = Formatear Lectura Correcta de Escanner
// -------------------------------------------------------------------------------------
// --- Incializalizamoms la lectura

      CALL  FILL
      ( BVAL    := #cero,
        RET_VAL := #retvalue,
        BLK     := "DB211_Lecturas_Scanner".Lec_Scanner[#NumScanner]
      );

      CALL  FILL
      ( BVAL    := #cero,
        RET_VAL := #retvalue,
        BLK     := "DB905_Estado_Escaners".Escaner[#NumScanner].Lectura
      );


      L     1;
      T     #CNT_Escritura;  // --- Inicializa el contador de caracteres de escritura
      L     11;
      T     #CNT_Lectura;
      L     0;
      T     #CNT_Datos_Pantalla;



      L     'N';
      T     "DB211_Lecturas_Scanner".Lec_Scanner[#NumScanner].Lectura_SCR[0];  //      Carga el primer caracter de la etiqueta existente



// -------------------------------------------------------------------------------------
// --- Bucle de lectura de Etiqueta

Inicio_bucle:NOP   0;  // --- INICIO BUCLE ETIQUETA
      L     #CNT_Escritura;
      L     #Numero_Caracteres;  //     Si estamos a la izquierda del primer Caracter ponemos la 'N'
      >=I;
      JC    Escribir_Etiqueta;  // --- Tomamos caracter de lectura de escaner ?


      L     #caracter_relleno;  // Nieves: modificación para que el JDT pueda truncar la lectura más facilmente   20/09/16
      T     "DB211_Lecturas_Scanner".Lec_Scanner[#NumScanner].Lectura_SCR[#CNT_Escritura];
      T     "DB905_Estado_Escaners".Escaner[#NumScanner].Lectura[#CNT_Datos_Pantalla];  // transfiero tambien al array temporal que nos hemos creado

      L     1;  // --- Incrementa contador caracteres
      L     #CNT_Datos_Pantalla;
      +I;
      T     #CNT_Datos_Pantalla;

      L     1;  // --- Incrementa contador caracteres
      L     #CNT_Escritura;
      +I;
      T     #CNT_Escritura;


// comprobación del caracter de escritura para no salirnos de rango
      SET;
      L     #CNT_Escritura;  // --- Mirar si se ha acabo la etiqueta
      L     "ROUT_Long_Etiqueta";
      <I;  // --- Si no llegamos al final repetimos el bucle
      JC    Inicio_bucle;

// si no hemos saltado es que hemos llegado al último caracter de escritura y tenemos que salir

      JU    Fin_Bucle;


// -------------------------------------------------------------------------------------
// -- Escribimos ahora la etiqueta

Escribir_Etiqueta:NOP   0;
      L     #Datos_E_Scanner[#CNT_Lectura];  // --- Leer carcater de la Etiqueta
      T     "DB211_Lecturas_Scanner".Lec_Scanner[#NumScanner].Lectura_SCR[#CNT_Escritura];  //     escribirlo en el registro de la etiqueta
      T     "DB905_Estado_Escaners".Escaner[#NumScanner].Lectura[#CNT_Datos_Pantalla];  // transfiero tambien al array temporal que nos hemos creado



// -------------------------------------------------------------------------------------
// -- incrementamos los contadores para pasar al siguiente caracter
siguiente_caracter:NOP   0;

      L     1;  // --- Incrementa contador caracteres
      L     #CNT_Escritura;
      +I;
      T     #CNT_Escritura;

      L     1;  // --- Incrementa contador caracteres
      L     #CNT_Lectura;
      +I;
      T     #CNT_Lectura;

      L     1;  // --- Incrementa contador caracteres
      L     #CNT_Datos_Pantalla;
      +I;
      T     #CNT_Datos_Pantalla;


      L     #CNT_Escritura;  // --- Mirar si se ha acabo la etiqueta
      L     "ROUT_Long_Etiqueta";
      <I;  // --- Si no llegamos al final repetimos el bucle
      JC    Inicio_bucle;

      JU    Fin_Bucle;  // --- Si termina la lectura correctamente cerramos protocolo



NETWORK
TITLE = Error lectura etiqueta no esperada
// -------------------------------------------------------------------------------------
// ---  Rellenar de error de etiqueta --> 'N000000000'

Error_lectura:NOP   0;

      L     1;  // --- Incializar CNT de Caracteres Escritos
      T     #CNT_Escritura;
      L     0;
      T     #CNT_Datos_Pantalla;


      L     'N';  // --- Caracter 'N'
      T     "DB211_Lecturas_Scanner".Lec_Scanner[#NumScanner].Lectura_SCR[0];


bucle_error:NOP   0;

      L     '0';  // --- Caracter '0'
      T     "DB211_Lecturas_Scanner".Lec_Scanner[#NumScanner].Lectura_SCR[#CNT_Escritura];
      T     "DB905_Estado_Escaners".Escaner[#NumScanner].Lectura[#CNT_Datos_Pantalla];


// -- incrementamos los contadores para desplazarnos en la estructura

      L     1;  // --- Incrementa contador caracteres
      L     #CNT_Escritura;
      +I;
      T     #CNT_Escritura;

      L     1;  // --- Incrementa contador caracteres
      L     #CNT_Datos_Pantalla;
      +I;
      T     #CNT_Datos_Pantalla;


      L     #CNT_Escritura;  // --- Mirar si se ha acabo la etiqueta
      L     "ROUT_Long_Etiqueta";
      <I;  // --- Si no llegamos al final repetimos el bucle ?
      JC    bucle_error;

      JU    Fin_Bucle;  // --- Si termina la lectura correctamente cerramos protocolo



NETWORK
TITLE = Confirmar al Scanner de leida la etiqueta
// -------------------------------------------------------------------------------------
// --- Confirmar al Scanner de leida la etiqueta

Fin_Bucle:NOP   0;

// -- Guardamos los datos de la etiqueta recogida en el DB

      L     #Datos_E_Scanner[3];  // --- Obtenemos un puntero al número de telegrama del Scanner
      T     QB [#PunteroSCR_A];  // --- Confirmamos la lectura con el número de telegrama del Scanner

      L     #Datos_E_Scanner[3];  // --- La lectura ha sido tratada anteriormente
      T     "DB214_CNT_Mens_SCR".RedScanners[#Numero_Red].CNT_NODO_PROF_SCR[#SCR_Actual];  //     Guardar el ID de la recepción y en el envio


      L     #CNT_LectCiclo;  // --- Incrementa el Numero de lecturas por ciclo
      L     1;
      +I;
      T     #CNT_LectCiclo;


NETWORK
TITLE = Actualizar datos pantalla
//===============================================================================================
//-- volcamos el dato del diagnóstico

      CALL  BLKMOV
      ( SRCBLK  := #Datos_Diagnostico,
        RET_VAL := #retvalue,
        DSTBLK  := "DB905_Estado_Escaners".Escaner[#NumScanner].Diagnostico
      );



//===============================================================================================


NETWORK
TITLE = salir de la funcion
// -------------------------------------------------------------------------------------
// --- Se sale de la función

Fin_funcion:NOP   0;

END_FUNCTION

FUNCTION "FC522_Buc_Busc_Etiquetas" : Void   // FC522, LAD
{ S7_Optimized_Access := 'FALSE' }
AUTHOR : ROUTER
NAME : 20130623
VERSION : 3.1
// stored: AutoNumber false, SetENOAutomatically false
   VAR_TEMP
      Valor_Etiqueta : ULInt;
      CNT_Scanner : UInt;
      CNT_Caracter_Etiqueta : UInt;
      Peso_caracter : ULInt;
      bucle_scanners : Bool;
      Fin_conversion : Bool;
      contador : UInt;
   END_VAR
BEGIN

REGION Network 1 (SCL)
   REGION inicializacion
       #Valor_Etiqueta := 0;
       #Peso_caracter := 1;
       #CNT_Caracter_Etiqueta := "ROUT_Long_Etiqueta" - 1;
       #CNT_Scanner := 1;
       #bucle_scanners := 1;
   END_REGION
END_REGION

REGION Network 2 (SCL)
   WHILE #bucle_scanners DO
       IF "DB211_Lecturas_Scanner".Lec_Scanner[#CNT_Scanner].Lectura_SCR[0] = 'N' THEN
           // convertir lectura iniciamos el bucle de conversión
           #contador := #CNT_Caracter_Etiqueta;
           #Valor_Etiqueta := 0;
           #Peso_caracter := 1;
           #Fin_conversion := 0;
           WHILE (NOT (#Fin_conversion)) DO
               IF (("DB211_Lecturas_Scanner".Lec_Scanner[#CNT_Scanner].Lectura_SCR[#contador] >= '0') AND ("DB211_Lecturas_Scanner".Lec_Scanner[#CNT_Scanner].Lectura_SCR[#contador] <= '9')) THEN
                   #Valor_Etiqueta += ((CHAR_TO_INT("DB211_Lecturas_Scanner".Lec_Scanner[#CNT_Scanner].Lectura_SCR[#contador])-48)* #Peso_caracter);
                   #contador -= 1;
                   #Peso_caracter *= 10;
               ELSE
                   #Fin_conversion := true;
                   "DB211_Lecturas_Scanner".Lec_Scanner[#CNT_Scanner].Lectura_SCR[0] := L#0;
                   // ya hemos terminado de convertir el valor, buscamos la etiqueta
              "FC716_Router_BuscarEtiqueta_Lint_y_sacar_orden"(Etiqueta := #Valor_Etiqueta,
                                                                    Numero_SCR := #CNT_Scanner);

               END_IF;

           END_WHILE;


       ELSE // pasar al siguiente scanenr
           #CNT_Scanner += 1;
           IF #CNT_Scanner <= "ROUT_Max_Scanners" THEN
               ;
           ELSE
               RETURN;
           END_IF;
       END_IF;
   END_WHILE;
END_REGION
END_FUNCTION

ORGANIZATION_BLOCK "OB121_PROG_ERR"   // OB121, LAD, ProgrammingError
TITLE = "Programming Error"
{ S7_Optimized_Access := 'FALSE' }
AUTHOR : ESTANDAR
VERSION : 3.0
// stored: SetENOAutomatically false
   VAR_TEMP
      OB121_EV_CLASS : Byte;   // 16#25, Event class 2, Entering event state, Internal fault event
      OB121_SW_FLT : Byte;   // 16#XX Software programming fault
      OB121_PRIORITY : Byte;   // Priority of OB Execution
      OB121_OB_NUMBR : Byte;   // 121 (Organization block 121, OB121)
      OB121_BLK_TYPE : Byte;   // 16#88/8A/8B/8C/8E Type of block fault occured in
      OB121_RESERVED_1 : Byte;   // Reserved for system
      OB121_FLT_REG : Word;   // 16#XX Specific register that caused fault
      OB121_BLK_NUM : Word;   // Number of block that programming fault occured in
      OB121_PRG_ADDR : Word;   // Address in block where programming fault occured
      OB121_DATE_TIME : Date_And_Time;   // Date and time OB121 started
   END_VAR
BEGIN
END_ORGANIZATION_BLOCK

ORGANIZATION_BLOCK "OB122_MOD_ERR"   // OB122, LAD, IOAccessError
TITLE = "Module Access Error"
{ S7_Optimized_Access := 'FALSE' }
AUTHOR : ESTANDAR
VERSION : 3.0
// stored: SetENOAutomatically false
   VAR_TEMP
      OB122_EV_CLASS : Byte;   // 16#29, Event class 2, Entering event state, Internal fault event
      OB122_SW_FLT : Byte;   // 16#XX Software error code
      OB122_PRIORITY : Byte;   // Priority of OB Execution
      OB122_OB_NUMBR : Byte;   // 122 (Organization block 122, OB122)
      OB122_BLK_TYPE : Byte;   // 16#88/8C/8E Type of block fault occured in
      OB122_MEM_AREA : Byte;   // Memory area where access error occured
      OB122_MEM_ADDR : Word;   // Memory address where access error occured
      OB122_BLK_NUM : Word;   // Block number in which error occured
      OB122_PRG_ADDR : Word;   // Program address where error occured
      OB122_DATE_TIME : Date_And_Time;   // Date and time OB1 started
   END_VAR
BEGIN
END_ORGANIZATION_BLOCK

ORGANIZATION_BLOCK "OB30_Interrupcion_Diag_profinet_ASi"   // OB30, LAD, CyclicInterrupt
{ S7_Optimized_Access := 'TRUE' }
// stored: SetENOAutomatically false
   VAR_INPUT
      Initial_Call : Bool;   // Initial call of this OB
      Event_Count : Int;   // Events discarded
   END_VAR
BEGIN

REGION Network 1: Diagnostico Red Profinet
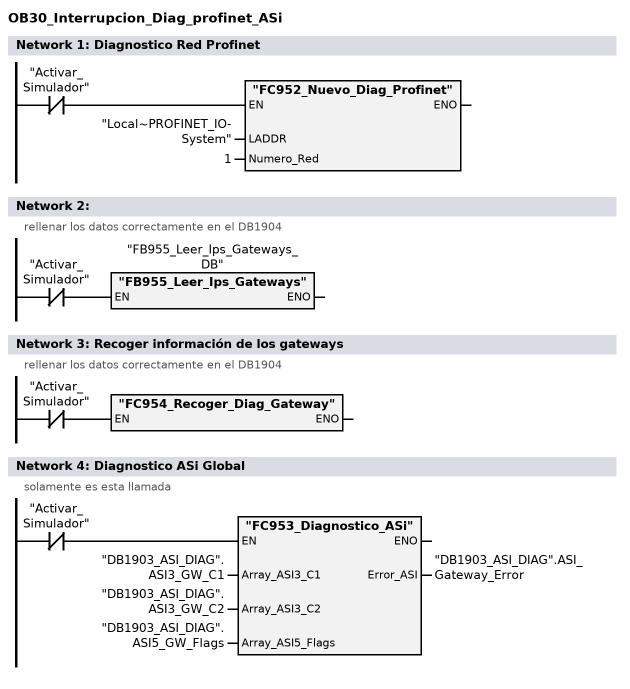
   RUNG wire#powerrail
      I_Contact( "Activar_Simulador" )
      "FC952_Nuevo_Diag_Profinet"(LADDR := "Local~PROFINET_IO-System", Numero_Red := 1)
   END_RUNG
   // the same network as SCL:
   IF NOT "Activar_Simulador" THEN
       "FC952_Nuevo_Diag_Profinet"(LADDR := "Local~PROFINET_IO-System", Numero_Red := 1);
   END_IF;
END_REGION

REGION Network 2
   // rellenar los datos correctamente en el DB1904
   RUNG wire#powerrail
      I_Contact( "Activar_Simulador" )
      "FB955_Leer_Ips_Gateways_DB"()
   END_RUNG
   // the same network as SCL:
   IF NOT "Activar_Simulador" THEN
       "FB955_Leer_Ips_Gateways_DB"();   // "FB955_Leer_Ips_Gateways"
   END_IF;
END_REGION

REGION Network 3: Recoger información de los gateways
   // rellenar los datos correctamente en el DB1904
   RUNG wire#powerrail
      I_Contact( "Activar_Simulador" )
      "FC954_Recoger_Diag_Gateway"()
   END_RUNG
   // the same network as SCL:
   IF NOT "Activar_Simulador" THEN "FC954_Recoger_Diag_Gateway"(); END_IF;
END_REGION

